	//BMS_CATL:
		(*gr_BMS_SOC						:=	gr_CATL_B2VST2SOC;
		gr_BMS_BatteryVoltage			:=	UINT_TO_REAL(gu16_CATL_B2TBMSHVVoltA);
		gr_BMS_Voltage					:=	UINT_TO_REAL(gu16_CATL_B2TBMSHVVoltA);
		//gr_BMS2_Voltage					:=	UINT_TO_REAL(gu16_CATL_B2TBMSHVVoltA);
		gs16_BMS_BatteryCurrent			:=	REAL_TO_INT(gr_CATL_B2VST2PackCurrent); 
		(*********)gu16_BMS_Maximum_Pack_Voltage	:=	REAL_TO_UINT(gr_CATL_B2VBI3PackAvaiMaxVolt); (*Limit applied to prevent overcharging*)
		gs16_BMS1_CCL					:=	REAL_TO_INT(gr_CATL_B2VAvailInpulseChrgCurr);
		gs16_BMS2_CCL					:=	REAL_TO_INT(gr_CATL_B2VAvailInpulseChrgCurr);
		//gu16_BMS_AverageCellVoltage		:=	(gu16_OrionBMS1_AverageCellVoltage + gu16_OrionBMS2_AverageCellVoltage) / 2;
		//gu16_BMS_LowCellVoltage			:=	MIN(gu16_OrionBMS1_LowCellVoltage, gu16_OrionBMS2_LowCellVoltage);
		//gu16_BMS_HighCellVoltage		:=	MAX(gu16_OrionBMS1_HighCellVoltage, gu16_OrionBMS2_HighCellVoltage);
		gr_BMS_AverageTemp				:=	INT_TO_REAL(g16_CATL_B2VST4AvgTemp);
		
		
		
		
		
	
		(*********)gu16_BMS1_LowCellmV		:=	REAL_TO_UINT(gr_CATL_B2VST5MinUcell*1000);
		//gu16_BMS2_LowCellmV		:=	gr_CATL_B2VST5MaxUcell*1000;
		(*********)gu16_BMS1_HighCellVoltage		:=	REAL_TO_UINT(gr_CATL_B2VST5MaxUcell);
		//gu16_BMS2_HighCellVoltage		:=	gu16_OrionBMS2_HighCellVoltage;
		//gu16_BMS1_LowCellVoltage_ID		:=	gu8_OrionBMS1_LowCellVoltNumber;
		//gu16_BMS2_LowCellVoltage_ID		:=	gu8_OrionBMS2_LowCellVoltNumber;
		//gu16_BMS1_HighCellVoltage_ID	:=	gu8_OrionBMS1_HighCellVoltNumber;
		//gu16_BMS2_HighCellVoltage_ID	:=	gu8_OrionBMS2_HighCellVoltNumber;	*)	
		
		
END_CASE




// First pass trigger resets charge interlock fault for plug release	
IF Main.firstPass.Q THEN
	chargeInterlockFlt := FALSE;
ELSIF gu16_OrionBMS1_FailsafeStatus.4 THEN
	chargeInterlockFlt := TRUE;
END_IF

END_PROGRAM

// Application/UserCode/Brusa/Brusa_1
(*==============================================================================================================*)
(*    Brusa charging function block calls and LED control                                                       *)
(*==============================================================================================================*)
PROGRAM Brusa_1
VAR
	Master           : BrusaControl; // Brusa charger master side
	Slave            : BrusaControl; // Brusa charger slave side
	
	LEDDem           : USINT; 
	LEDState         : BYTE;         // Case variable for LED states
	
	M_StateDem       : USINT;
	S_StateDem       : USINT;
	M_Unlock         : BOOL;
	S_Unlock         : BOOL;
	M_ErrCLr         : BOOL;
	S_ErrClr         : BOOL;
	M_ChargeStopAct  : BOOL;
	M_DCHVCurrLimMax : REAL;
	S_DCHVCurrLimMax : REAL;
	M_ACCurrLimMax   : REAL;
	S_ACCurrLimMax   : REAL;
	M_DCHVVoltLimMax : REAL;
	S_DCHVVoltLimMax : REAL;
	M_BalancingAmps  : REAL := 2;
	S_BalancingAmps  : REAL := 2;

	PulseTmr         : WORD;	
	PulseLength      : WORD := 50;    // Initialised to 500ms (50 * 10ms scans)
	Pulsing          : BOOL := FALSE;
	
	chargeStatus     : BYTE;
END_VAR
VAR CONSTANT
(*Charger statuswords =========================================================================================*)
	NLG_STATUS_CHARGE		: BYTE	:= 4;
	
(*Charger controlwords ========================================================================================*)
	NLG_CONTROL_STANDBY		: BYTE	:= 0;
	NLG_CONTROL_CHARGE		: BYTE	:= 1;
	
(*NLG LED States ==============================================================================================*)
	LED_OFF			        : BYTE	:= 0;
	LED_RED					: BYTE	:= 2;
	LED_GREEN_PULSE	        : BYTE  := 3;
	LED_GREEN				: BYTE	:= 4;
	LED_BLUE		        : BYTE	:= 8;
	LED_BLUE_GREEN_PULSE	: BYTE	:= 11;
	
(*Charge status  ==============================================================================================*)
	NOT_CONNECTED           : BYTE  := 0;
	STOPPED                 : BYTE  := 1;
	ERROR_ACTIVE            : BYTE  := 2;
	BALANCING               : BYTE  := 3;
	FULLY_CHARGED           : BYTE  := 4;
	NO_AC                   : BYTE  := 5;
	CHARGING                : BYTE  := 6;
	
END_VAR

(*==============================================================================================================*)
(*    Brusa charging function block calls                                                                       *)
(*==============================================================================================================*)
 // FreeContactor(); // Uncomment this to pulse welded contactors


Master (                Master := TRUE, // Master charger
	                 	BMS_OK := (OrionBMS1_RxConversion.Safety_OK OR OrionBMS2_RxConversion.Safety_OK),
                  CtrlPilotDet := Brusa1_Rx.S_CtrlPilotDet,
                  ProximityDet := Brusa1_Rx.S_ProximityDet,
                         Error := Brusa1_Rx.S_Err,
                         ACDet := Brusa1_Rx.S_ACDet,
               BalancingActive := OrionBMS1_RxConversion.gq_BMS1_BalActive,
                      SysState := gu8_SystemState,
                      StateAct := Brusa1_Rx.StateAct,
                        Status := Brusa1_Rx.StatusPP,
                Balancing_Amps := MAX	(2,(HMI_Rx.RAW_Pack_1_Balancing_Amps * 0.1)),
         Offset_Charge_Voltage := MAX	(4,(HMI_Rx.RAW_Pack_1_Offset_Volts    * 0.1)),
                           CCL := gs16_BMS1_CCL,
		      MaxChargingVolts := OrionBMS1_RxConversion.gr_OrionBMS1_Max_Charging_Voltage,
			     StopChargeReq := HMI_Rx.StopChargeRq,
			 ReportedMaxACCurr := Brusa1_Rx.ACCurrMaxAct_Rx,
			         CPMaxAmps := Brusa1_Rx.ACCurrMaxCP_Rx,
						   
                      StateDem => M_StateDem,
				  StopCharging => ,
                        Unlock => M_Unlock,
                 ErrorClearOut => M_ErrCLr,
                DCHVCurrLimMax => M_DCHVCurrLimMax,
                  ACCurrLimMax => M_ACCurrLimMax,
                DCHVVoltLimMax => M_DCHVVoltLimMax );
						   
						   
Slave (                 Master := FALSE, // Slave charger
	                 BMS_OK := (OrionBMS1_RxConversion.Safety_OK OR OrionBMS2_RxConversion.Safety_OK),
                  CtrlPilotDet := Brusa1_Rx.S_CtrlPilotDet,
                  ProximityDet := Brusa1_Rx.S_ProximityDet,
                         Error := Brusa2_Rx.S_Err,
                         ACDet := Brusa2_Rx.S_ACDet,
               BalancingActive := OrionBMS2_RxConversion.gq_BMS2_BalActive,
                      SysState := gu8_SystemState,
                      StateAct := Brusa2_Rx.StateAct,
                        Status := Brusa1_Rx.StatusPP,
                Balancing_Amps := MAX	(2,(HMI_Rx.RAW_Pack_2_Balancing_Amps * 0.1)),
         Offset_Charge_Voltage := MAX	(4,(HMI_Rx.RAW_Pack_2_Offset_Volts    * 0.1)),
                           CCL := gs16_BMS2_CCL,
			  MaxChargingVolts := OrionBMS2_RxConversion.gr_OrionBMS2_Max_Charging_Voltage,
			     StopChargeReq := HMI_Rx.StopChargeRq,
             ReportedMaxACCurr := Brusa2_Rx.ACCurrMaxAct_Rx,
			 	     CPMaxAmps := Brusa1_Rx.ACCurrMaxCP_Rx,
						   
                      StateDem => S_StateDem,
                        //Unlock => S_Unlock,
                 ErrorClearOut => S_ErrCLr,
                DCHVCurrLimMax => S_DCHVCurrLimMax,
                  ACCurrLimMax => S_ACCurrLimMax,
                DCHVVoltLimMax => S_DCHVVoltLimMax);	

(*==============================================================================================================*)
(*    Brusa LED control                                                                                         *)
(*==============================================================================================================*)

// Check to see if the charger is plugged in
IF (gu8_SystemState = PLUGIN_SYS) THEN    
            
	// Check for any errors
	IF (gu8_SystemState = ERROR_SYS) THEN             
		LEDDem := LED_RED;
		chargeStatus := 1;
	
	// Check for fully charged
	ELSIF gq_BattFullyCharged THEN                                                       
		LEDDem := LED_GREEN;
	
	// Check to see if charging is active
	ELSIF ((Brusa1_Rx.StateAct = NLG_STATUS_CHARGE) OR (Brusa2_Rx.StateAct = NLG_STATUS_CHARGE)) THEN
		
		// Check to see if balancing is active (Only if charging is also active)
		IF (OrionBMS1_RxConversion.gq_BMS1_BalActive OR OrionBMS2_RxConversion.gq_BMS2_BalActive) THEN
			LEDDem := LED_BLUE_GREEN_PULSE;
		ELSE
			LEDDem := LED_BLUE;
		END_IF
		
	// Check to see that AC is detected
	ELSIF NOT (Brusa1_Rx.S_ACDet) THEN
		LEDDem := LED_GREEN_PULSE; 

END_IF

ELSE 
LEDDem := 0; // OFF 

END_IF

(*==============================================================================================================*)
(*    Charge status for HMI Tx                                                                                  *)
(*==============================================================================================================*)

// System is in error state
IF (gu8_SystemState = ERROR_SYS) THEN
	chargeStatus := ERROR_ACTIVE;

// System is in plug in state (charge plug detected)
ELSIF (gu8_SystemState = PLUGIN_SYS) THEN
	
	// Charge stopped by HMI
	IF (M_ChargeStopAct) THEN
		chargeStatus := STOPPED;
	
	// Vehicle is fully charged	
	ELSIF (BMSData.Batteries_Fully_Charged AND NOT (OrionBMS1_RxConversion.gq_BMS1_BalActive OR OrionBMS2_RxConversion.gq_BMS2_BalActive)) THEN
		chargeStatus := FULLY_CHARGED;
	
	// Waiting for AC	
	ELSIF NOT (Brusa1_Rx.S_ACDet AND Brusa2_Rx.S_ACDet) THEN
		chargeStatus := NO_AC; 
	
	// BMS is balancing	
	ELSIF (OrionBMS1_RxConversion.gq_BMS1_BalActive OR OrionBMS2_RxConversion.gq_BMS2_BalActive) THEN
		chargeStatus := BALANCING;
	
	// Vehicle is charging	
	ELSIF ((Brusa1_Rx.StateAct = NLG_STATUS_CHARGE) OR (Brusa2_Rx.StateAct = NLG_STATUS_CHARGE)) THEN
		chargeStatus := CHARGING;
		
	END_IF
	
// Charge plug not detected	
ELSE
	chargeStatus := NOT_CONNECTED;

END_IF

ACTION FreeContactor:
(*==============================================================================================================*)
(*    Uncomment this action to pulse the contactor free                                                         *)
(*==============================================================================================================*)
Pulsing := TRUE;                                               // Flag to stop Contactor control from running (main())

PulseTmr := PulseTmr + 1;                                      // Increment pulse timer every scan

IF (PulseTmr = PulseLength) THEN                               // Pulse length is number of 10ms scans
DO_q_Battery1ChargeMain_DO := NOT DO_q_Battery1ChargeMain_DO;  // Switch output
PulseTmr := 0;                                                 // Reset timer
END_IF
END_ACTION

END_PROGRAM

// Application/UserCode/Brusa/BrusaControl_1
(*===================================================================================================*)
(* Charger Control                                                                                   *)
(*===================================================================================================*)
FUNCTION_BLOCK BrusaControl_1
VAR_INPUT
(*Variable inputs ===================================================================================*)
	Master                  : BOOL;             // Master?
	BMS_OK     			    : BOOL;             // Battery safety ok signal
	CtrlPilotDet            : BOOL;
	ProximityDet            : BOOL;
	Error                   : BOOL;             // Brusa error
	ACDet                   : BOOL;
	BalancingActive         : BOOL; 
	StopChargeReq           : BOOL;             // Request to stop charging
	SysState                : BYTE;             // System state
	StateAct                : BYTE;             // Brusa recieved state
	Status                  : BYTE;             // Status PP?
	Balancing_Amps          : REAL;
	OffSet_Charge_Voltage   : REAL;
	CCL                     : REAL;
	MaxChargingVolts        : REAL;             // Max charging voltage from BMS
	ReportedMaxACCurr       : WORD;             // Reported AC max current from Brusa
	CPMaxAmps               : UINT;             // Control pilot allowable current
	
	
	
END_VAR
VAR_OUTPUT
	StateDem		        : USINT;           // Charger state request
	Unlock                  : BOOL;            // Charger unlock
	ErrorClearOut           : BOOL := FALSE;   // Request error clear
	StopCharging            : BOOL;            // Latch for stop charging request
	DCHVCurrLimMax			: REAL := 0;
	ACCurrLimMax			: REAL := 0;
	DCHVVoltLimMax			: REAL := 0;

END_VAR

VAR
	ChargerStates           :	tUpdate;         // Charger state machine variable
	
	ResetCnt                :   BYTE;            // Number of reset attempts

	ChargeDelayTmr          :   WORD;            // Scan counter to delay start charging 
	
	ResetOK     			:	BOOL;            // OK to reset
	
	CurrentLimit            :   REAL;            // Maximum allowable current
			
END_VAR

VAR CONSTANT

(*Charger control words ============================================================================*)
	NLG_CONTROL_STANDBY		:	USINT	:=	0;    // Standby request
	NLG_CONTROL_CHARGE		:	USINT	:=	1;	  // Charge request
	NLG_CONTROL_SLEEP		:	USINT	:=	6;    // Sleep request
	NLG_CONTROL_SNA			:	USINT	:=	7;    
	
(*Charger status words =============================================================================*)
	NLG_STATUS_SLEEP		:	USINT	:=	0;
	NLG_STATUS_WAKEUP		:	USINT	:=	1;
	NLG_STATUS_STANDBY		:	USINT	:=	2;
	NLG_STATUS_READY2CHARGE	:	USINT	:=	3;
	NLG_STATUS_CHARGE		:	USINT	:=	4;
	NLG_STATUS_SHUTDOWN		:	USINT	:=	5;
	
(* Case step constants =============================================================================*)
	_Sleep                  :   BYTE    := 0;
	_Standby                :   BYTE 	:= 1;
	_Charging               :   BYTE    := 2;
	_Error                  :   BYTE    := 255;
	
(* Charger plug in states ==========================================================================*)
	CHARGER_DETECTED		:	BYTE	:=	0;
	CHARGER_NOTCONNECTED	:	BYTE	:=	5;
	
	PP_32A					:	BYTE	:=	3;
	PP_64A					:	BYTE	:=	4;
	
END_VAR

(*===================================================================================================*)
(* Charger state machine                                                                             *)
(*===================================================================================================*)

// Discuss error clearing - looks like error clear message is always set to false

(* Handle charge lock request =======================================================================*)	
IF (StopChargeReq) THEN                        // Move to standy if charge stop requested from HMI
	StopCharging := TRUE;
ELSIF (StopCharging AND NOT ProximityDet) THEN // Only allow charging once the charge plug has been removed and reinserted
	StopCharging := FALSE;
END_IF

CASE ChargerStates.Step OF
(* Sleep state ======================================================================================*)	
_Sleep:
	
	Unlock := TRUE;                           // Unlock charge plug

	IF (StateAct <> 0) THEN                   // Moved out of sleep state into wakeup state
		ChargerStates.Next := _Standby;       // Move to standby state 
	END_IF
	
(* Standby state ====================================================================================*)	
_Standby:
		
	Unlock := TRUE;                                          // Unlock charge plug
		
	IF OkToCharge() THEN                                     // Charging conditions OK (If charging conditions are met then lock should engage automatically)
		Unlock := FALSE;                                     // Allow charger to lock
		IF (StateAct = NLG_STATUS_READY2CHARGE) OR (StateAct = NLG_STATUS_CHARGE) THEN
		ChargerStates.Next := _Charging;                     // Move to charging state
		END_IF
	ELSIF (Error) THEN
		ChargerStates.Next := _Error;                        // Move to error state
	ELSIF (StateAct = NLG_STATUS_SLEEP) THEN
		ChargerStates.Next := _Sleep;                        // Move to sleep state
	ELSE
		StateDem :=	NLG_CONTROL_STANDBY;                     // Set STANDBY state
	END_IF
	
(* Charging state ===================================================================================*)
_Charging:
	
	StateDem :=	NLG_CONTROL_CHARGE;          // Set CHARGING state 

	IF NOT (OkToCharge()) THEN               // If not ok to charge check for errors
		
		IF (Error) THEN
			ChargerStates.Next := _Error;    // Move to error state 
		ELSE
			ChargerStates.Next := _Standby;  // Move back to standby state 
		END_IF
		
	END_IF
	
(* Error state ======================================================================================*)
_Error:

		IF (OkToReset()) THEN	
			
			ErrorClearOut := SEL((ChargerStates.Tmr < 100), FALSE, TRUE); // Request error clear
			
			IF (ChargerStates.Tmr > 6000) THEN   // 1 min - charger requires 1 min to attempt automatic recovery or temp recovery
				ResetCnt   := ResetCnt +1;       // Increment reset count
				ChargerStates.Next := _Standby;  // Move back to Standby state	
			END_IF
			
		END_IF	
	
END_CASE

(*Set the DC current limit depending on balancing status ==========================================*)
DCHVCurrLimMax := SEL( BalancingActive, CCL, MIN(CCL, Balancing_Amps));

(*Set the AC current limit based on the wire that is plugged in ===================================*)
IF (Brusa1_Rx.ACCurrMaxPP = PP_32A) THEN
	CurrentLimit	:=	MIN(15, ((CPMaxAmps/20)-1));    // Div by 200 to get single side and A from mA, then -1 for lead acid battery
ELSIF (Brusa1_Rx.ACCurrMaxPP = PP_64A) THEN
	CurrentLimit	:=	MIN(28, ((CPMaxAmps/20)-1));    // Div by 200 to get single side and A from mA, then -1 for lead acid battery
ELSE
	CurrentLimit	:=	0;
END_IF

(* Delay charge and then ramp current up to max - Add 50mA each scan ==============================*)

// If available currrent limit drops then drop requested current immediately
IF (ACCurrLimMax > CurrentLimit) THEN
	ACCurrLimMax := CurrentLimit;
	
// If available current is less than requested increase by 50mA each scan (e.g. 30Amps achieved in 6s)
ELSIF (ACCurrLimMax < CurrentLimit) THEN
	ACCurrLimMax := ACCurrLimMax + 0.005;

// Otherwise request the maximum allowable current
ELSE
	ACCurrLimMax := CurrentLimit;
END_IF

(* Limit maximum voltage to be delivered to each pack =============================================*)
DCHVVoltLimMax	:=	(MaxChargingVolts) - (OffSet_Charge_Voltage); 

Update(ADR(ChargerStates));                                     // State machine update

(*===================================================================================================*)
(* Monitor charging conditions                                                                       *)
(*===================================================================================================*)
METHOD OkToCharge : BOOL
VAR_INPUT
END_VAR
(*===================================================================================================*)
(* Monitor charging conditions                                                                       *)
(*===================================================================================================*)
OkToCharge := ((BMS_OK                                 	                               AND  // Check BMS safety is OK
              (CtrlPilotDet OR ACDet)                                                  AND  // Check for Control pilot or ACHV
	        //(ProximityDet                                                            AND  // Check plug proximity detect
			  (Status = CHARGER_DETECTED)                                              AND  // Check staus charger detected
			   NOT (Error OR StopChargeReq OR StopCharging)));                              // Check there are no errors or stop charge request
END_METHOD

(*===================================================================================================*)
(* Monitor reset conditions                                                                          *)
(*===================================================================================================*)
METHOD OkToReset : BOOL
VAR_INPUT
END_VAR
(*===================================================================================================*)
(* Monitor reset conditions                                                                          *)
(*===================================================================================================*)

OkToReset := ((StateAct = NLG_STATUS_STANDBY) AND   // Check for standby mode
			  (ResetCnt < 3));                      // Check reset count is less than 3
END_METHOD

END_FUNCTION_BLOCK

// Application/UserCode/CAN1/CAN1_Rx_1
PROGRAM CAN1_Rx_1
VAR
	Accelerator_Dennis_Rx	:	Receive_CAN1_EXD_28bit;
	Brake_Dennis_Rx			:	Receive_CAN1_EXD;
	GearSelect_Dennis_Rx	:	Receive_CAN1_EXD_28bit;
	AirPressure_Dennis_Rx	:	Receive_CAN1_EXD;
	
	EBC1_KB_Rx				:	Receive_CAN1_EXD;
	VDC1_KB_Rx				:	Receive_CAN1_EXD;
	EBC2_KB_Rx				:	Receive_CAN1_EXD;
	
	RegenStick01_Rx			:	Receive_CAN1_EXD;
	RegenStick12_Rx			:	Receive_CAN1_EXD;
	
	Bob_Handbrake_Rx	:	Receive_CAN1_EXD;
	Bob_Brake_Rx		:	Receive_CAN1_EXD;
	Bob_Accel_Rx		:	Receive_CAN1_EXD;
	Bob_RegenSelector_Rx	:	Receive_CAN1_EXD;
	
	Bob_WheelSpeed_Rx	:	Receive_CAN1_EXD_28bit;
	Bob_J1939_AirPressure_Rx	:	Receive_CAN1_EXD;
	
	Temperature_Rx		:	Receive_CAN1_EXD;
	Dennis_StabTracDisable_Rx	:	Receive_CAN1_EXD;
	
	Accelerator_Dennis_Rx_Timer	:	TON;
	Brake_Dennis_Rx_Timer		:	TON;
	GearSelect_Dennis_Rx_Timer	:	TON;
	Airpressure_Dennis_Rx_Timer	:	TON;
	
	hq_Bob_RightDrive_Compromised	: BOOL;
	hq_Bob_LeftDrive_Compromised	: BOOL;
	hq_Bob_RightFront_Compromised	: BOOL;
	hq_Bob_LeftFront_Compromised	: BOOL;
	
	Merc_AIR1_EAPU		:	Receive_CAN1_EXD;
	MercStalk_Rx: Receive_CAN1_EXD;
	Merc_Neutral_CAN1: BOOL := FALSE;
	Merc_Drive_CAN1: BOOL := FALSE;
	Merc_Reverse_CAN1: BOOL := FALSE;
	Dennis_No_Press: BOOL;
	Dennis_Up: BOOL;
	Dennis_Down: BOOL;
	LOADCTU: BOOL;
	InitialiseCounterValue: BYTE;
END_VAR

{region "Message Rx check"}
Accelerator_Dennis_Rx	(u32_COBID	:=	16#0CFF0211,
						q_NewData => ,
						au8_Data => ,
						u8_Length => 			);
				
(*Brake_Dennis_Rx	(u32_COBID	:=	16#18F0010B,
				q_NewData => ,
				au8_Data => ,
				u8_Length => 			);*)
				
GearSelect_Dennis_Rx	(u32_COBID	:=	16#0C010305,
						q_NewData => ,
						au8_Data => ,
						u8_Length => 			);
						
AirPressure_Dennis_Rx	(u32_COBID	:=	16#18FEAE30,
						q_NewData => ,
						au8_Data => ,
						u8_Length => 			);
						
EBC1_KB_Rx				(u32_COBID	:=	16#18F0010B,
						q_NewData => ,
						au8_Data => ,
						u8_Length => 			);

VDC1_KB_Rx				(u32_COBID	:=	16#18FE4F0B,
						q_NewData => ,
						au8_Data => ,
						u8_Length => 			);

EBC2_KB_Rx				(u32_COBID	:=	16#18FEBF0B,
						q_NewData => ,
						au8_Data => ,
						u8_Length => 			);
						
RegenStick01_Rx			(u32_COBID	:=	16#18F00021,
						q_NewData => ,
						au8_Data => ,
						u8_Length => 			);
							 
RegenStick12_Rx			(u32_COBID	:=	16#0C000003,
						q_NewData => ,
						au8_Data => ,
						u8_Length => 			);
							 
Bob_Handbrake_Rx(u32_COBID	:=	16#18FF0447,
			q_NewData => ,
			au8_Data => ,
			u8_Length => 			);
				 
Bob_Brake_Rx(u32_COBID	:=	16#14FF010B,
			q_NewData => ,
			au8_Data => ,
			u8_Length => 			);
				 
Bob_Accel_Rx(u32_COBID	:=	16#10F00300,
			q_NewData => ,
			au8_Data => ,
			u8_Length => 			);
				 
Bob_RegenSelector_Rx(u32_COBID	:=	16#14FF0300,
			q_NewData => ,
			au8_Data => ,
			u8_Length => 			);
				 
Bob_WheelSpeed_Rx(u32_COBID	:=	16#08FE6E0B,
			q_NewData => ,
			au8_Data => ,
			u8_Length => 			);
				 
Bob_J1939_AirPressure_Rx(u32_COBID := 16#14FEAE17,
			q_NewData => ,
			au8_Data => ,
			u8_Length => 			);
				 
Temperature_Rx(u32_COBID := 16#18FF12C4,
			q_NewData => ,
			au8_Data => ,
			u8_Length => 			);
				 
Dennis_StabTracDisable_Rx(u32_COBID := 16#18FE4F0B,
			q_NewData => ,
			au8_Data => ,
			u8_Length => 			);
				 
MercStalk_Rx	(u32_COBID	:=	16#18FF0400,
						q_NewData => ,
						au8_Data => ,
						u8_Length => 			);
(*Moved to CAN 3*)
Merc_AIR1_EAPU(u32_COBID := 16#14FEAE30,
		 	q_NewData => ,
			au8_Data => ,
			u8_Length =>			);			

{endregion}
Merc_Neutral_CAN1			:=	MercStalk_Rx.au8_Data[4].0;
Merc_Drive_CAN1				:=	MercStalk_Rx.au8_Data[4].1;
Merc_Reverse_CAN1			:=	MercStalk_Rx.au8_Data[4].2;
{region "Assign data to receive variables"}		
gu8_AccelPedal_Dennis_Rx	:=	Accelerator_Dennis_Rx.au8_Data[3];
gq_Dennis_Accel_NewData		:=	Accelerator_Dennis_Rx.q_NewData;				

gq_BrakePedal_Dennis_Rx		:=	Brake_Dennis_Rx.au8_Data[0].6;
gu8_BrakePedal_Perc_Dennis_Rx	:=	Brake_Dennis_Rx.au8_Data[1];

gu8_GearSelector_Dennis_Rx	:=	GearSelect_Dennis_Rx.au8_Data[2];
	 // Dennis Regen Select
		  
	InitialiseCounterValue := InitialiseCounterValue + 1;
	IF InitialiseCounterValue > 250 THEN
	InitialiseCounterValue := 201;
	END_IF
				   
 	IF GearSelect_Dennis_Rx.au8_Data[2] = 224 THEN
	Dennis_No_Press := TRUE;
	ELSE
	Dennis_No_Press := FALSE;
	END_IF
	
	IF GearSelect_Dennis_Rx.au8_Data[2] = 249 THEN
	Dennis_Up	:= TRUE;
	ELSE
	Dennis_Up := FALSE;
	END_IF
	
	IF GearSelect_Dennis_Rx.au8_Data[2] = 247 THEN
	Dennis_Down	:= TRUE;
	ELSE
	Dennis_Down := FALSE;
	END_IF
		 
	IF Dennis_Regen.DennisRegen.CV > 4 OR InitialiseCounterValue < 200 THEN 
	LOADCTU := TRUE;
	ELSE
	LOADCTU := FALSE;
	END_IF 
//		  
IF (AirPressure_Dennis_Rx.au8_Data[2] > 0 OR AirPressure_Dennis_Rx.au8_Data[3] > 0) THEN
	gu8_Dennis_AirPressureBrake1_Rx	:=	AirPressure_Dennis_Rx.au8_Data[2];
	gu8_Dennis_AirPressureBrake2_Rx	:=	AirPressure_Dennis_Rx.au8_Data[3];
	gu8_Dennis_AirPressureSusp_Rx	:=	AirPressure_Dennis_Rx.au8_Data[5];
END_IF

	 
gu8_EBC1_ASREngineControlActive				:=BOOL_TO_USINT(EBC1_KB_Rx.au8_Data[0].0) + SHL(BOOL_TO_USINT(EBC1_KB_Rx.au8_Data[0].1), 1);
gu8_EBC1_ASRBrakeControlActive				:=BOOL_TO_USINT(EBC1_KB_Rx.au8_Data[0].2) + SHL(BOOL_TO_USINT(EBC1_KB_Rx.au8_Data[0].3), 1);
gu8_EBC1_ABSActive							:=BOOL_TO_USINT(EBC1_KB_Rx.au8_Data[0].4) + SHL(BOOL_TO_USINT(EBC1_KB_Rx.au8_Data[0].5), 1);
gu8_EBC1_EBSBrakeSwitch						:=BOOL_TO_USINT(EBC1_KB_Rx.au8_Data[0].6) + SHL(BOOL_TO_USINT(EBC1_KB_Rx.au8_Data[0].7), 1);
gu8_EBC1_BrakePedalPosition					:=EBC1_KB_Rx.au8_Data[1];
gu8_EBC1_ABSOffroadSwitch					:=BOOL_TO_USINT(EBC1_KB_Rx.au8_Data[2].0) + SHL(BOOL_TO_USINT(EBC1_KB_Rx.au8_Data[2].1), 1);
gu8_EBC1_ASROffroadSwitch					:=BOOL_TO_USINT(EBC1_KB_Rx.au8_Data[2].2) + SHL(BOOL_TO_USINT(EBC1_KB_Rx.au8_Data[2].3), 1);
gu8_EBC1_ASRHillholderSwitch				:=BOOL_TO_USINT(EBC1_KB_Rx.au8_Data[2].4) + SHL(BOOL_TO_USINT(EBC1_KB_Rx.au8_Data[2].5), 1);
gu8_EBC1_TractionControlOverrideSwtich		:=BOOL_TO_USINT(EBC1_KB_Rx.au8_Data[2].6) + SHL(BOOL_TO_USINT(EBC1_KB_Rx.au8_Data[2].7), 1);
gu8_EBC1_AcceleratorInterlockSwitch			:=BOOL_TO_USINT(EBC1_KB_Rx.au8_Data[3].0) + SHL(BOOL_TO_USINT(EBC1_KB_Rx.au8_Data[3].1), 1);
gu8_EBC1_EngineDerateSwitch					:=BOOL_TO_USINT(EBC1_KB_Rx.au8_Data[3].2) + SHL(BOOL_TO_USINT(EBC1_KB_Rx.au8_Data[3].3), 1);
gu8_EBC1_EngineAuxiliaryShutdownSwitch		:=BOOL_TO_USINT(EBC1_KB_Rx.au8_Data[3].4) + SHL(BOOL_TO_USINT(EBC1_KB_Rx.au8_Data[3].5), 1);
gu8_EBC1_RemoteAcceleratorEnableSwitch		:=BOOL_TO_USINT(EBC1_KB_Rx.au8_Data[3].6) + SHL(BOOL_TO_USINT(EBC1_KB_Rx.au8_Data[3].7), 1);
gu8_EBC1_EngineRetarderSelection			:=EBC1_KB_Rx.au8_Data[4];
gu8_EBC1_ABSFullyOperational				:=BOOL_TO_USINT(EBC1_KB_Rx.au8_Data[5].0) + SHL(BOOL_TO_USINT(EBC1_KB_Rx.au8_Data[5].1), 1);
gu8_EBC1_gu8_EBC1_EBSRedWarningSignal		:=BOOL_TO_USINT(EBC1_KB_Rx.au8_Data[5].2) + SHL(BOOL_TO_USINT(EBC1_KB_Rx.au8_Data[5].3), 1);
gu8_EBC1_ABSEBSAmberWarningSignal			:=BOOL_TO_USINT(EBC1_KB_Rx.au8_Data[5].4) + SHL(BOOL_TO_USINT(EBC1_KB_Rx.au8_Data[5].5), 1);
gu8_EBC1_ATCASRInformationSignal			:=BOOL_TO_USINT(EBC1_KB_Rx.au8_Data[5].6) + SHL(BOOL_TO_USINT(EBC1_KB_Rx.au8_Data[5].7), 1);
gu8_EBC1_SrcAddrOfCrtllingDevForBrkCtrl		:=EBC1_KB_Rx.au8_Data[6];
gu8_EBC1_HaltBrakeSwitch					:=BOOL_TO_USINT(EBC1_KB_Rx.au8_Data[7].2) + SHL(BOOL_TO_USINT(EBC1_KB_Rx.au8_Data[7].3), 1);
gu8_EBC1_TrailerABSStatus					:=BOOL_TO_USINT(EBC1_KB_Rx.au8_Data[7].4) + SHL(BOOL_TO_USINT(EBC1_KB_Rx.au8_Data[7].5), 1);
gu8_EBC1_TractorMntdTrailerABSWarningSignal	:=BOOL_TO_USINT(EBC1_KB_Rx.au8_Data[7].6) + SHL(BOOL_TO_USINT(EBC1_KB_Rx.au8_Data[7].7), 1);

gu16_EBC2_KB_FrontAxleSpeed_Rx		:=	USINT_TO_UINT(EBC2_KB_Rx.au8_Data[0]) + SHL(USINT_TO_UINT(EBC2_KB_Rx.au8_Data[1]), 8);
gu16_EBC2_KB_FrontLeftRelSpd_Rx		:=	EBC2_KB_Rx.au8_Data[2];
gu16_EBC2_KB_FrontRightRelSpd_Rx	:=	EBC2_KB_Rx.au8_Data[3];
gu16_EBC2_KB_RearLeft1RelSpd_Rx		:=	EBC2_KB_Rx.au8_Data[4];
gu16_EBC2_KB_RearRight1RelSpd_Rx	:=	EBC2_KB_Rx.au8_Data[5];
gu16_EBC2_KB_RearLeft2RelSpd_Rx		:=	EBC2_KB_Rx.au8_Data[6];
gu16_EBC2_KB_RearRight2RelSpd_Rx	:=	EBC2_KB_Rx.au8_Data[7];

gu8_RegenStick01Pos					:=	RegenStick01_Rx.au8_Data[0];
gu8_RegenStick12Pos					:=	RegenStick12_Rx.au8_Data[0];	
	 
(*	 
VDC1_KB_Rx.au8_Data[0];
VDC1_KB_Rx.au8_Data[1];
VDC1_KB_Rx.au8_Data[2];
VDC1_KB_Rx.au8_Data[3];
VDC1_KB_Rx.au8_Data[4];
VDC1_KB_Rx.au8_Data[5];
VDC1_KB_Rx.au8_Data[6];
VDC1_KB_Rx.au8_Data[7];
*)		

gq_Bob_Handbrake_CAN	:=	Bob_Handbrake_Rx.au8_Data[0].0;
gu8_Bob_BrakePos_CAN	:=	Bob_Brake_Rx.au8_Data[1];
	
gu8_Bob_Accel_CAN		:=	Bob_Accel_Rx.au8_Data[1];
gu8_Bob_RegenSelector_CAN	:=	Bob_RegenSelector_Rx.au8_Data[4];
	
IF (Bob_WheelSpeed_Rx.au8_Data[0] <> 254 AND Bob_WheelSpeed_Rx.au8_Data[1] <> 254) THEN
	gu16_Bob_RightDrive_CAN	:=	USINT_TO_UINT(Bob_WheelSpeed_Rx.au8_Data[0]) + SHL(USINT_TO_UINT(Bob_WheelSpeed_Rx.au8_Data[1]), 8);
	hq_Bob_RightDrive_Compromised := FALSE;
ELSE
	IF (hq_Bob_LeftDrive_Compromised = FALSE) THEN
		gu16_Bob_RightDrive_CAN := gu16_Bob_LeftDrive_CAN;
	ELSIF (hq_Bob_RightFront_Compromised = FALSE) THEN
		gu16_Bob_RightDrive_CAN := gu16_Bob_RightFront_CAN;
	ELSIF (hq_Bob_LeftFront_Compromised = FALSE) THEN
		gu16_Bob_RightDrive_CAN := gu16_Bob_LeftFront_CAN;
	ELSE
		gu16_Bob_RightDrive_CAN := 0;
	END_IF
	hq_Bob_RightDrive_Compromised := TRUE;
END_IF
IF (Bob_WheelSpeed_Rx.au8_Data[2] <> 254 AND Bob_WheelSpeed_Rx.au8_Data[3] <> 254) THEN
	gu16_Bob_LeftDrive_CAN	:=	USINT_TO_UINT(Bob_WheelSpeed_Rx.au8_Data[2]) + SHL(USINT_TO_UINT(Bob_WheelSpeed_Rx.au8_Data[3]), 8);
	hq_Bob_LeftDrive_Compromised := FALSE;
ELSE
	IF (hq_Bob_RightDrive_Compromised = FALSE) THEN
		gu16_Bob_LeftDrive_CAN := gu16_Bob_RightDrive_CAN;
	ELSIF (hq_Bob_RightFront_Compromised = FALSE) THEN
		gu16_Bob_LeftDrive_CAN := gu16_Bob_RightFront_CAN;
	ELSIF (hq_Bob_LeftFront_Compromised = FALSE) THEN
		gu16_Bob_LeftDrive_CAN := gu16_Bob_LeftFront_CAN;
	ELSE
		gu16_Bob_LeftDrive_CAN := 0;
	END_IF
	hq_Bob_LeftDrive_Compromised := TRUE;
END_IF
IF (Bob_WheelSpeed_Rx.au8_Data[4] <> 254 AND Bob_WheelSpeed_Rx.au8_Data[5] <> 254) THEN
	gu16_Bob_RightFront_CAN	:=	USINT_TO_UINT(Bob_WheelSpeed_Rx.au8_Data[4]) + SHL(USINT_TO_UINT(Bob_WheelSpeed_Rx.au8_Data[5]), 8);
	hq_Bob_RightFront_Compromised := FALSE;
ELSE
	IF (hq_Bob_RightDrive_Compromised = FALSE) THEN
		gu16_Bob_RightFront_CAN := gu16_Bob_RightDrive_CAN;
	ELSIF (hq_Bob_LeftDrive_Compromised = FALSE) THEN
		gu16_Bob_RightFront_CAN := gu16_Bob_LeftDrive_CAN;
	ELSIF (hq_Bob_LeftFront_Compromised = FALSE) THEN
		gu16_Bob_RightFront_CAN := gu16_Bob_LeftFront_CAN;
	ELSE
		gu16_Bob_RightFront_CAN := 0;
	END_IF
	hq_Bob_RightFront_Compromised := TRUE;
END_IF
IF (Bob_WheelSpeed_Rx.au8_Data[6] <> 254 AND Bob_WheelSpeed_Rx.au8_Data[7] <> 254) THEN
	gu16_Bob_LeftFront_CAN	:=	USINT_TO_UINT(Bob_WheelSpeed_Rx.au8_Data[6]) + SHL(USINT_TO_UINT(Bob_WheelSpeed_Rx.au8_Data[7]), 8);
	hq_Bob_LeftFront_Compromised := FALSE;
ELSE
	IF (hq_Bob_RightDrive_Compromised = FALSE) THEN
		gu16_Bob_LeftFront_CAN := gu16_Bob_RightDrive_CAN;
	ELSIF (hq_Bob_LeftDrive_Compromised = FALSE) THEN
		gu16_Bob_LeftFront_CAN := gu16_Bob_LeftDrive_CAN;
	ELSIF (hq_Bob_RightFront_Compromised = FALSE) THEN
		gu16_Bob_LeftFront_CAN := gu16_Bob_RightFront_CAN;
	ELSE
		gu16_Bob_LeftFront_CAN := 0;
	END_IF
	hq_Bob_LeftFront_Compromised := TRUE;
END_IF
	 
IF (hq_Bob_RightDrive_Compromised = TRUE OR
	hq_Bob_LeftDrive_Compromised = TRUE OR
	hq_Bob_RightFront_Compromised = TRUE OR
	hq_Bob_LeftFront_Compromised = TRUE ) THEN

	gq_Bob_WheelSpeedSensor_Fail := TRUE;
ELSE
	gq_Bob_WheelSpeedSensor_Fail := FALSE;
END_IF

gu8_Bob_ServiceBrakeAirPressCircuit1_CAN	:=	Bob_J1939_AirPressure_Rx.au8_Data[2];
gu8_Bob_ServiceBrakeAirPressCircuit2_CAN	:=	Bob_J1939_AirPressure_Rx.au8_Data[3];
gu8_Bob_AirSuspensionSupplyPress_CAN		:=	Bob_J1939_AirPressure_Rx.au8_Data[5];
gq_Bob_AirCompressorStatus_CAN				:=	Bob_J1939_AirPressure_Rx.au8_Data[6].0;

		 
(*Temperature_Rx.au8_Data[0];*)
	 
IF (gu8_ChassisType = CHASSIS_DENNIS) THEN
	(*gq_StabTracDisable_Rx	:=	Dennis_StabTracDisable_Rx.au8_Data[0].3;*)
	gq_StabTracDisable_Rx	:=	USINT_TO_BOOL(gu8_EBC1_ASROffroadSwitch);
ELSIF (gu8_ChassisType = CHASSIS_BOB OR gu8_ChassisType = CHASSIS_ESTARGLIDER) THEN
	gq_StabTracDisable_Rx	:=	Bob_Brake_Rx.au8_Data[4].2;
END_IF
				  
{endregion}
	 
{region "Comms Loss Check"}
Accelerator_Dennis_Rx_Timer(IN := NOT(Accelerator_Dennis_Rx.q_NewData), PT := T#3S);
Brake_Dennis_Rx_Timer(IN := NOT(EBC1_KB_Rx.q_NewData), PT := T#3S);
GearSelect_Dennis_Rx_Timer(IN := NOT(GearSelect_Dennis_Rx.q_NewData), PT := T#3S);
Airpressure_Dennis_Rx_Timer(IN := NOT(Airpressure_Dennis_Rx.q_NewData), PT := T#3S);
IF (Accelerator_Dennis_Rx_Timer.Q = TRUE AND Brake_Dennis_Rx_Timer.Q = TRUE AND
	GearSelect_Dennis_Rx_Timer.Q = TRUE AND Airpressure_Dennis_Rx_Timer.Q = TRUE) THEN
	gq_Dennis_CAN1_CommsLoss	:=	TRUE;
ELSE
	gq_Dennis_CAN1_CommsLoss	:=	FALSE;
END_IF
{endregion}
	 

gu8_Merc_AirComepressor_Rq	:=	BOOL_TO_USINT(Merc_AIR1_EAPU.au8_Data[6].0) + SHL(BOOL_TO_USINT(Merc_AIR1_EAPU.au8_Data[6].1), 1);
IF ((*gu8_Merc_AirComepressor_Rq*)gq_Bob_AirCompressorStatus_CAN = TRUE(*1*)) THEN
	gq_Merc_AirComp_Rq := TRUE;
ELSE
	gq_Merc_AirComp_Rq := FALSE;
END_IF	
	 
CAN1_RxConversion();

END_PROGRAM

// Application/UserCode/CAN1/CAN1_RxConversion_1
PROGRAM CAN1_RxConversion_1
VAR
END_VAR
VAR CONSTANT
	NEUTRAL	:	USINT	:=	16#7D;
	DRIVE	:	USINT	:=	16#FC;
	REVERSE	:	USINT	:=	16#DF;
	
	AIRPRESSURE_CF	:	REAL	:=	0.08;
	
	FRONTAXLESPEED_CF	:	REAL	:=	0.00390625;
	RELATIVESPEED_CF	:	REAL	:=	0.0625;
	RELATIVESPEED_OFFSET	:	REAL	:=	-7.8125;
END_VAR


IF  gu8_GearSelector_Dennis_Rx = NEUTRAL AND gq_BrakeSwitch AND gr_VehicleSpeed_kmph <1 AND gr_VehicleSpeed_kmph >-1 THEN
	gq_Neutral_Dennis_Rq	:=	TRUE;
	gq_Drive_Dennis_Rq		:=	FALSE;
	gq_Reverse_Dennis_Rq	:=	FALSE;
ELSIF gu8_GearSelector_Dennis_Rx = DRIVE AND gq_BrakeSwitch AND gr_VehicleSpeed_kmph > -1 THEN
	gq_Neutral_Dennis_Rq	:=	FALSE;
	gq_Drive_Dennis_Rq		:=	TRUE;
	gq_Reverse_Dennis_Rq	:=	FALSE;
ELSIF gu8_GearSelector_Dennis_Rx = REVERSE AND gq_BrakeSwitch AND gr_VehicleSpeed_kmph < 1 THEN
	gq_Neutral_Dennis_Rq	:=	FALSE;
	gq_Drive_Dennis_Rq		:=	FALSE;
	gq_Reverse_Dennis_Rq	:=	TRUE;
ELSE
	;
END_IF
	
IF (gu8_EBC1_ABSActive = 1) THEN
	gq_ABSActive	:=	TRUE;
ELSE
	gq_ABSActive	:=	FALSE;
END_IF

	
gr_EBC2_KB_FrontAxleSpeed				:=	gu16_EBC2_KB_FrontAxleSpeed_Rx * FRONTAXLESPEED_CF;
gr_EBC2_KB_FrontLeftRelSpd				:=	gu16_EBC2_KB_FrontLeftRelSpd_Rx * RELATIVESPEED_CF + RELATIVESPEED_OFFSET;
gr_EBC2_KB_FrontRightRelSpd				:=	gu16_EBC2_KB_FrontRightRelSpd_Rx * RELATIVESPEED_CF + RELATIVESPEED_OFFSET;
gr_EBC2_KB_RearLeft1RelSpd				:=	gu16_EBC2_KB_RearLeft1RelSpd_Rx * RELATIVESPEED_CF + RELATIVESPEED_OFFSET;
gr_EBC2_KB_RearRight1RelSpd				:=	gu16_EBC2_KB_RearRight1RelSpd_Rx * RELATIVESPEED_CF + RELATIVESPEED_OFFSET;
gr_EBC2_KB_RearLeft2RelSpd				:=	gu16_EBC2_KB_RearLeft2RelSpd_Rx * RELATIVESPEED_CF + RELATIVESPEED_OFFSET;
gr_EBC2_KB_RearRight2RelSpd				:=	gu16_EBC2_KB_RearRight2RelSpd_Rx * RELATIVESPEED_CF + RELATIVESPEED_OFFSET;
		

gr_Bob_Accel	:=	(USINT_TO_REAL(gu8_Bob_Accel_CAN) / 250);
IF (gu8_Bob_BrakePos_CAN > 0) THEN
	gq_Bob_Brake_CAN	:=	TRUE;
ELSE
	gq_Bob_Brake_CAN	:=	FALSE;
END_IF

gr_Bob_ServiceBrakeAirPressCircuit1		:=	gu8_Bob_ServiceBrakeAirPressCircuit1_CAN * AIRPRESSURE_CF;
gr_Bob_ServiceBrakeAirPressCircuit2		:=	gu8_Bob_ServiceBrakeAirPressCircuit2_CAN * AIRPRESSURE_CF;
gr_Bob_AirSuspensionSupplyPress			:=	gu8_Bob_AirSuspensionSupplyPress_CAN * AIRPRESSURE_CF;

END_PROGRAM

// Application/UserCode/CAN1/CAN1_TCMs_Tx_1
PROGRAM CAN1_TCMs_Tx_1
VAR
	(*TCM ECR*)
	ht_RCM_C01_Tx	:	EPEC_CANVXD.Msg;
	ht_RCM_C02_Tx	:	EPEC_CANVXD.Msg;
	ht_TCM_C01_Tx	:	EPEC_CANVXD.Msg;
	ht_TCM_C02_Tx	:	EPEC_CANVXD.Msg;
	ht_TCM_C03_Tx	:	EPEC_CANVXD.Msg;
	ht_TCM_C05_Tx	:	EPEC_CANVXD.Msg;
	ht_TCM_C06_Tx	:	EPEC_CANVXD.Msg;
	ht_TCM_C08_Tx	:	EPEC_CANVXD.Msg;
	ht_TCM_C10_Tx	:	EPEC_CANVXD.Msg;
	ht_TCM_C11_Tx	:	EPEC_CANVXD.Msg;
	ht_TCM_C22_Tx	:	EPEC_CANVXD.Msg;
	ht_TCM_DM1_Tx	:	EPEC_CANVXD.Msg;
	ht_TRF1_TCM_Tx	:	EPEC_CANVXD.Msg;
	
	ht_MCM_C01_Tx	:	EPEC_CANVXD.Msg;
	ht_MCM_C02_Tx	:	EPEC_CANVXD.Msg;
	ht_MCM_C03_Tx	:	EPEC_CANVXD.Msg;
	ht_MCM_C07_Tx	:	EPEC_CANVXD.Msg;
	ht_MCM_C10_Tx	:	EPEC_CANVXD.Msg;
	ht_MCM_C14_Tx	:	EPEC_CANVXD.Msg;
	ht_MCM_C15_Tx	:	EPEC_CANVXD.Msg;
	ht_MCM_C23_Tx	:	EPEC_CANVXD.Msg;
	
	ht_Compressor_Status	:	EPEC_CANVXD.Msg;
	
	hu8_C01_Checksum	:	USINT;
	hu8_C02_Checksum	:	USINT;
	hu8_C03_Checksum	:	USINT;
	hu8_C05_Checksum	:	USINT;
	hu8_C08_Checksum	:	USINT;
	hu8_C10_Checksum	:	USINT;
	hu8_C11_Checksum	:	USINT;
	hu8_M23_Checksum	:	USINT;
	
	hu8_4BitMessageCounter10ms		:	USINT;
	hu8_4BitMessageCounter20ms		:	USINT;
	hu8_4BitMessageCounter50ms		:	USINT;
	hu8_4BitMessageCounter100ms		:	USINT;
	
	hq_CycleAlternator	:	BOOL;
	hton_MessageSend50ms_Timer	:	TON;
	hton_MessageSend_Timer		:	TON;
	Tx_Timer	:	TON;
	ClutchEnaged: BOOL;
END_VAR
VAR CONSTANT
	MAX_REGEN_TORQUE	:	UINT	:=	4090;
END_VAR
VAR
	ClutchStatB: BOOL := TRUE;
	ClutchStatA: BOOL := TRUE;
	ClutchEngaged: BOOL;
	ClutchIntermediate: BOOL;
	ClutchDisengaged: BOOL;
	TONIntermediate: TON;
END_VAR

ht_RCM_C01_Tx.ID		:=	16#CFF000F OR EPEC_CANVXD.MASK_29BIT;
ht_RCM_C01_Tx.Data[0]	:=	16#FF;
ht_RCM_C01_Tx.Data[1].0	:=	gq_RegenActive;
ht_RCM_C01_Tx.Data[1].1	:=	0;
ht_RCM_C01_Tx.Data[1].2	:=	gq_RegenActive;
ht_RCM_C01_Tx.Data[1].3	:=	0;
ht_RCM_C01_Tx.Data[1].4	:=	1;
ht_RCM_C01_Tx.Data[1].5	:=	1;
ht_RCM_C01_Tx.Data[1].6	:=	1;
ht_RCM_C01_Tx.Data[1].7	:=	1;
ht_RCM_C01_Tx.Data[2]	:=	16#FF;
ht_RCM_C01_Tx.Data[3]	:=	REAL_TO_USINT(ABS(MIN(0, gr_MCU_TorqueCommand_PreCF * BOOL_TO_USINT(gq_RegenActive) / 20))); //Should be 0 when not regenning and then a positive value when it is doing so
ht_RCM_C01_Tx.Data[4]	:=	REAL_TO_USINT(MAX_REGEN_TORQUE / 20); //Maximum regen torque is 4090Nm (MCU CAN Protocol v4.1)
ht_RCM_C01_Tx.Data[5]	:=	16#FF;
ht_RCM_C01_Tx.Data[6]	:=	16#FF;
ht_RCM_C01_Tx.Data[7]	:=	16#FF;
ht_RCM_C01_Tx.Len		:=	8;
	 
ht_RCM_C02_Tx.ID		:=	16#14FF000F OR EPEC_CANVXD.MASK_29BIT;
ht_RCM_C02_Tx.Data[0]	:=	16#FF;
ht_RCM_C02_Tx.Data[1]	:=	16#FF;
ht_RCM_C02_Tx.Data[2]	:=	16#FF;
ht_RCM_C02_Tx.Data[3]	:=	16#FF;
ht_RCM_C02_Tx.Data[4]	:=	16#FF;
ht_RCM_C02_Tx.Data[5]	:=	16#FF;
ht_RCM_C02_Tx.Data[6]	:=	16#FF;
ht_RCM_C02_Tx.Data[7]	:=	16#FF;
ht_RCM_C02_Tx.Len		:=	8;
	 
ht_TCM_C01_Tx.ID		:=	16#08FF0003 OR EPEC_CANVXD.MASK_29BIT;
ht_TCM_C01_Tx.Data[0]	:=	16#FF;
ht_TCM_C01_Tx.Data[1]	:=	16#FF;
ht_TCM_C01_Tx.Data[2]	:=	16#FF;
ht_TCM_C01_Tx.Data[3]	:=	16#FF;
ht_TCM_C01_Tx.Data[4]	:=	16#FF;
ht_TCM_C01_Tx.Data[5]	:=	16#FF;
ht_TCM_C01_Tx.Data[6].0	:=	1;
ht_TCM_C01_Tx.Data[6].1	:=	1;
ht_TCM_C01_Tx.Data[6].2	:=	1;
ht_TCM_C01_Tx.Data[6].3	:=	1;
ht_TCM_C01_Tx.Data[6].4	:=	hu8_4BitMessageCounter10ms.0;
ht_TCM_C01_Tx.Data[6].5	:=	hu8_4BitMessageCounter10ms.1;
ht_TCM_C01_Tx.Data[6].6	:=	hu8_4BitMessageCounter10ms.2;
ht_TCM_C01_Tx.Data[6].7	:=	hu8_4BitMessageCounter10ms.3;
hu8_C01_Checksum		:=	16#FF - (ht_TCM_C01_Tx.Data[0] + ht_TCM_C01_Tx.Data[1] + ht_TCM_C01_Tx.Data[2] + ht_TCM_C01_Tx.Data[3] + ht_TCM_C01_Tx.Data[4] + ht_TCM_C01_Tx.Data[5] + ht_TCM_C01_Tx.Data[6]);;
ht_TCM_C01_Tx.Data[7]	:=	hu8_C01_Checksum;
ht_TCM_C01_Tx.Len		:=	8;

ht_TCM_C02_Tx.ID		:=	16#08FF0103 OR EPEC_CANVXD.MASK_29BIT;
ht_TCM_C02_Tx.Data[0]	:=	16#FF;
ht_TCM_C02_Tx.Data[1]	:=	16#FF;
ht_TCM_C02_Tx.Data[2]	:=	UINT_TO_USINT(gu16_TCM2_OutputShaftSpeed);
ht_TCM_C02_Tx.Data[3]	:=	UINT_TO_USINT(SHR(gu16_TCM2_OutputShaftSpeed, 8));
ht_TCM_C02_Tx.Data[4]	:=	16#FF;
ht_TCM_C02_Tx.Data[5].0	:=	gu8_TCM2_DrvDirec_Stat.0;
ht_TCM_C02_Tx.Data[5].1	:=	gu8_TCM2_DrvDirec_Stat.1;
ht_TCM_C02_Tx.Data[5].2	:=	1;
ht_TCM_C02_Tx.Data[5].3	:=	1;
ht_TCM_C02_Tx.Data[5].4	:=	gu8_TCM2_RotSens_Stat.0;
ht_TCM_C02_Tx.Data[5].5	:=	gu8_TCM2_RotSens_Stat.1;
ht_TCM_C02_Tx.Data[5].6	:=	1;
ht_TCM_C02_Tx.Data[5].7	:=	1;
ht_TCM_C02_Tx.Data[6].0	:=	ClutchStatA;
ht_TCM_C02_Tx.Data[6].1	:=	ClutchStatB;
ht_TCM_C02_Tx.Data[6].2	:=	1;
ht_TCM_C02_Tx.Data[6].3	:=	1;
ht_TCM_C02_Tx.Data[6].4	:=	hu8_4BitMessageCounter10ms.0;
ht_TCM_C02_Tx.Data[6].5	:=	hu8_4BitMessageCounter10ms.1;
ht_TCM_C02_Tx.Data[6].6	:=	hu8_4BitMessageCounter10ms.2;
ht_TCM_C02_Tx.Data[6].7	:=	hu8_4BitMessageCounter10ms.3;
hu8_C02_Checksum	:=	16#FF - (ht_TCM_C02_Tx.Data[0] + ht_TCM_C02_Tx.Data[1] + ht_TCM_C02_Tx.Data[2] + ht_TCM_C02_Tx.Data[3] + ht_TCM_C02_Tx.Data[4] + ht_TCM_C02_Tx.Data[5] + ht_TCM_C02_Tx.Data[6]);
ht_TCM_C02_Tx.Data[7]	:=	hu8_C02_Checksum;
ht_TCM_C02_Tx.Len		:=	8;

ht_TCM_C03_Tx.ID		:=	16#08FF0203 OR EPEC_CANVXD.MASK_29BIT;
ht_TCM_C03_Tx.Data[0]	:=	16#FF;
ht_TCM_C03_Tx.Data[1]	:=	16#FF;
ht_TCM_C03_Tx.Data[2]	:=	UINT_TO_USINT(gu16_TCM03_ShaftSpeed_Tx);
ht_TCM_C03_Tx.Data[3]	:=	UINT_TO_USINT(SHR(gu16_TCM03_ShaftSpeed_Tx, 8));
ht_TCM_C03_Tx.Data[4]	:=	16#FF;
ht_TCM_C03_Tx.Data[5]	:=	16#FF;
ht_TCM_C03_Tx.Data[6].0	:=	1;
ht_TCM_C03_Tx.Data[6].1	:=	1;
ht_TCM_C03_Tx.Data[6].2	:=	1;
ht_TCM_C03_Tx.Data[6].3	:=	1;
ht_TCM_C03_Tx.Data[6].4	:=	hu8_4BitMessageCounter10ms.0;
ht_TCM_C03_Tx.Data[6].5	:=	hu8_4BitMessageCounter10ms.1;
ht_TCM_C03_Tx.Data[6].6	:=	hu8_4BitMessageCounter10ms.2;
ht_TCM_C03_Tx.Data[6].7	:=	hu8_4BitMessageCounter10ms.3;
hu8_C03_Checksum	:=	16#FF - (ht_TCM_C03_Tx.Data[0] + ht_TCM_C03_Tx.Data[1] + ht_TCM_C03_Tx.Data[2] + ht_TCM_C03_Tx.Data[3] + ht_TCM_C03_Tx.Data[4] + ht_TCM_C03_Tx.Data[5] + ht_TCM_C03_Tx.Data[6]);
ht_TCM_C03_Tx.Data[7]	:=	hu8_C03_Checksum;
ht_TCM_C03_Tx.Len		:=	8;

ht_TCM_C05_Tx.ID		:=	16#14FF0403 OR EPEC_CANVXD.MASK_29BIT;
ht_TCM_C05_Tx.Data[0]	:=	16#FF;
ht_TCM_C05_Tx.Data[1]	:=	16#FF;
ht_TCM_C05_Tx.Data[2]	:=	16#FF;
ht_TCM_C05_Tx.Data[3]	:=	16#FF;
ht_TCM_C05_Tx.Data[4]	:=	16#FF;
ht_TCM_C05_Tx.Data[5]	:=	16#FF;
ht_TCM_C05_Tx.Data[6].0	:=	gq_Gear_Neutral;
ht_TCM_C05_Tx.Data[6].1	:=	0;
ht_TCM_C05_Tx.Data[6].2	:=	1;
ht_TCM_C05_Tx.Data[6].3	:=	1;
ht_TCM_C05_Tx.Data[6].4	:=	hu8_4BitMessageCounter100ms.0;
ht_TCM_C05_Tx.Data[6].5	:=	hu8_4BitMessageCounter100ms.1;
ht_TCM_C05_Tx.Data[6].6	:=	hu8_4BitMessageCounter100ms.2;
ht_TCM_C05_Tx.Data[6].7	:=	hu8_4BitMessageCounter100ms.3;
hu8_C05_Checksum	:=	16#FF - (ht_TCM_C05_Tx.Data[0] + ht_TCM_C05_Tx.Data[1] + ht_TCM_C05_Tx.Data[2] + ht_TCM_C05_Tx.Data[3] + ht_TCM_C05_Tx.Data[4] + ht_TCM_C05_Tx.Data[5] + ht_TCM_C05_Tx.Data[6]);
ht_TCM_C05_Tx.Data[7]	:=	hu8_C05_Checksum;
ht_TCM_C05_Tx.Len		:=	8;

ht_TCM_C06_Tx.ID		:=	16#18FF0503 OR EPEC_CANVXD.MASK_29BIT;
ht_TCM_C06_Tx.Data[0]	:=	16#FF;
ht_TCM_C06_Tx.Data[1]	:=	16#FF;
ht_TCM_C06_Tx.Data[2]	:=	16#FF;
ht_TCM_C06_Tx.Data[3]	:=	16#FF;
ht_TCM_C06_Tx.Data[4]	:=	16#FF;
ht_TCM_C06_Tx.Data[5]	:=	16#FF;
ht_TCM_C06_Tx.Data[6]	:=	16#FF;
ht_TCM_C06_Tx.Data[7]	:=	16#FF;
ht_TCM_C06_Tx.Len		:=	8;

ht_TCM_C08_Tx.ID		:=	16#0CFF0703 OR EPEC_CANVXD.MASK_29BIT;
ht_TCM_C08_Tx.Data[0]	:=	16#FF;
ht_TCM_C08_Tx.Data[1]	:=	16#FF;
ht_TCM_C08_Tx.Data[2]	:=	16#FF;
ht_TCM_C08_Tx.Data[3]	:=	16#FF;
ht_TCM_C08_Tx.Data[4]	:=	gu8_TCM8_Gear;
ht_TCM_C08_Tx.Data[5]	:=	16#FF;
ht_TCM_C08_Tx.Data[6].0	:=	NOT(gq_Gear_Neutral);
ht_TCM_C08_Tx.Data[6].1	:=	0;
ht_TCM_C08_Tx.Data[6].2	:=	gu8_TCM8_DrvDirByGr_Stat.0;
ht_TCM_C08_Tx.Data[6].3	:=	gu8_TCM8_DrvDirByGr_Stat.1;
ht_TCM_C08_Tx.Data[6].4	:=	hu8_4BitMessageCounter20ms.0;
ht_TCM_C08_Tx.Data[6].5	:=	hu8_4BitMessageCounter20ms.1;
ht_TCM_C08_Tx.Data[6].6	:=	hu8_4BitMessageCounter20ms.2;
ht_TCM_C08_Tx.Data[6].7	:=	hu8_4BitMessageCounter20ms.3;
hu8_C08_Checksum	:=	16#FF - (ht_TCM_C08_Tx.Data[0] + ht_TCM_C08_Tx.Data[1] + ht_TCM_C08_Tx.Data[2] + ht_TCM_C08_Tx.Data[3] + ht_TCM_C08_Tx.Data[4] + ht_TCM_C08_Tx.Data[5] + ht_TCM_C08_Tx.Data[6]);
ht_TCM_C08_Tx.Data[7]	:=	hu8_C08_Checksum;
ht_TCM_C08_Tx.Len		:=	8;

ht_TCM_C10_Tx.ID		:=	16#10FF0903 OR EPEC_CANVXD.MASK_29BIT;
ht_TCM_C10_Tx.Data[0]	:=	16#FF;
ht_TCM_C10_Tx.Data[1]	:=	16#FF;
ht_TCM_C10_Tx.Data[2]	:=	16#FF;
ht_TCM_C10_Tx.Data[3]	:=	16#FF;
ht_TCM_C10_Tx.Data[4]	:=	16#FF;
ht_TCM_C10_Tx.Data[5]	:=	16#FF;
ht_TCM_C10_Tx.Data[6].0	:=	1;
ht_TCM_C10_Tx.Data[6].1	:=	1;
ht_TCM_C10_Tx.Data[6].2	:=	1;
ht_TCM_C10_Tx.Data[6].3	:=	1;
ht_TCM_C10_Tx.Data[6].4	:=	hu8_4BitMessageCounter50ms.0;
ht_TCM_C10_Tx.Data[6].5	:=	hu8_4BitMessageCounter50ms.1;
ht_TCM_C10_Tx.Data[6].6	:=	hu8_4BitMessageCounter50ms.2;
ht_TCM_C10_Tx.Data[6].7	:=	hu8_4BitMessageCounter50ms.3;
hu8_C10_Checksum	:=	16#FF - (ht_TCM_C10_Tx.Data[0] + ht_TCM_C10_Tx.Data[1] + ht_TCM_C10_Tx.Data[2] + ht_TCM_C10_Tx.Data[3] + ht_TCM_C10_Tx.Data[4] + ht_TCM_C10_Tx.Data[5] + ht_TCM_C10_Tx.Data[6]);
ht_TCM_C10_Tx.Data[7]	:=	0;
ht_TCM_C10_Tx.Len		:=	8;

ht_TCM_C11_Tx.ID		:=	16#08FF0303 OR EPEC_CANVXD.MASK_29BIT;
ht_TCM_C11_Tx.Data[0]	:=	gu8_TCM8_Gear;
ht_TCM_C11_Tx.Data[1]	:=	16#FF;
ht_TCM_C11_Tx.Data[2]	:=	16#FF;
ht_TCM_C11_Tx.Data[3]	:=	16#FF;
ht_TCM_C11_Tx.Data[4]	:=	16#FF;
ht_TCM_C11_Tx.Data[5]	:=	16#FF;
ht_TCM_C11_Tx.Data[6]	:=	UINT_TO_USINT(gu16_TCM11_ActualGearRatio);
ht_TCM_C11_Tx.Data[7]	:=	UINT_TO_USINT(SHR(gu16_TCM11_ActualGearRatio, 8));
ht_TCM_C11_Tx.Len		:=	8;

ht_TCM_C22_Tx.ID		:=	16#18FF0703 OR EPEC_CANVXD.MASK_29BIT;
ht_TCM_C22_Tx.Data[0]	:=	16#FF;
ht_TCM_C22_Tx.Data[1]	:=	16#FF;
ht_TCM_C22_Tx.Data[2]	:=	16#FF;
ht_TCM_C22_Tx.Data[3]	:=	16#FF;
ht_TCM_C22_Tx.Data[4]	:=	16#FF;
ht_TCM_C22_Tx.Data[5]	:=	16#FF;
ht_TCM_C22_Tx.Data[6]	:=	16#FF;
ht_TCM_C22_Tx.Data[7]	:=	16#FF;
ht_TCM_C22_Tx.Len		:=	8;

(*Message not sent*)
ht_TCM_DM1_Tx.ID		:=	16#10FECA03 OR EPEC_CANVXD.MASK_29BIT;
ht_TCM_DM1_Tx.Data[0]	:=	0;
ht_TCM_DM1_Tx.Data[1]	:=	0;
ht_TCM_DM1_Tx.Data[2]	:=	0;
ht_TCM_DM1_Tx.Data[3]	:=	0;
ht_TCM_DM1_Tx.Data[4]	:=	0;
ht_TCM_DM1_Tx.Data[5]	:=	0;
ht_TCM_DM1_Tx.Data[6]	:=	0;
ht_TCM_DM1_Tx.Data[7]	:=	0;
ht_TCM_DM1_Tx.Len		:=	8;

ht_TRF1_TCM_Tx.ID		:=	16#18FEF803 OR EPEC_CANVXD.MASK_29BIT;
ht_TRF1_TCM_Tx.Data[0]	:=	16#FF;
ht_TRF1_TCM_Tx.Data[1]	:=	16#FF;
ht_TRF1_TCM_Tx.Data[2]	:=	16#FF;
ht_TRF1_TCM_Tx.Data[3]	:=	16#FF;
ht_TRF1_TCM_Tx.Data[4]	:=	16#FF;
ht_TRF1_TCM_Tx.Data[5]	:=	16#FF;
ht_TRF1_TCM_Tx.Data[6]	:=	16#FF;
ht_TRF1_TCM_Tx.Data[7]	:=	16#FF;
ht_TRF1_TCM_Tx.Len		:=	8;

(*********************************************************************)
ht_MCM_C01_Tx.ID		:=	16#08FF0001 OR EPEC_CANVXD.MASK_29BIT;
ht_MCM_C01_Tx.Data[0]	:=	16#FF;
ht_MCM_C01_Tx.Data[1]	:=	16#FF;
ht_MCM_C01_Tx.Data[2]	:=	16#FF;
ht_MCM_C01_Tx.Data[3]	:=	16#FF;
ht_MCM_C01_Tx.Data[4]	:=	16#FF;
ht_MCM_C01_Tx.Data[5]	:=	16#FF;
ht_MCM_C01_Tx.Data[6]	:=	16#FF;
ht_MCM_C01_Tx.Data[7]	:=	16#FF;
ht_MCM_C01_Tx.Len		:=	8;

ht_MCM_C02_Tx.ID		:=	16#08FF0101 OR EPEC_CANVXD.MASK_29BIT; (*commented out due to already being sent*)
ht_MCM_C02_Tx.Data[0]	:=	BOOL_TO_USINT(DOS_q_BatteryDischargeMain_DO);
ht_MCM_C02_Tx.Data[1]	:=	16#FF;
ht_MCM_C02_Tx.Data[2]	:=	UINT_TO_USINT(gu16_MCM02_EngineTorque_Tx);
ht_MCM_C02_Tx.Data[3]	:=	UINT_TO_USINT(SHR(gu16_MCM02_EngineTorque_Tx, 8));
ht_MCM_C02_Tx.Data[4]	:=	UINT_TO_USINT(gu16_RPM_Display);
ht_MCM_C02_Tx.Data[5]	:=	UINT_TO_USINT(SHR(gu16_RPM_Display, 8));
ht_MCM_C02_Tx.Data[6]	:=	16#FF;
ht_MCM_C02_Tx.Data[7]	:=	16#FF;
ht_MCM_C02_Tx.Len		:=	8;

ht_MCM_C03_Tx.ID		:=	16#14FF0001 OR EPEC_CANVXD.MASK_29BIT;
ht_MCM_C03_Tx.Data[0]	:=	16#FF;
ht_MCM_C03_Tx.Data[1]	:=	16#FF;
ht_MCM_C03_Tx.Data[2]	:=	16#FF;
ht_MCM_C03_Tx.Data[3]	:=	16#FF;
ht_MCM_C03_Tx.Data[4]	:=	16#FF;
ht_MCM_C03_Tx.Data[5]	:=	16#FF;
ht_MCM_C03_Tx.Data[6]	:=	16#FF;
ht_MCM_C03_Tx.Data[7]	:=	16#FF;
ht_MCM_C03_Tx.Len		:=	8;

ht_MCM_C07_Tx.ID		:=	16#14FF0401 OR EPEC_CANVXD.MASK_29BIT;
ht_MCM_C07_Tx.Data[0]	:=	16#FF;
ht_MCM_C07_Tx.Data[1]	:=	16#FF;
ht_MCM_C07_Tx.Data[2]	:=	16#FF;
ht_MCM_C07_Tx.Data[3]	:=	16#FF;
ht_MCM_C07_Tx.Data[4]	:=	16#FF;
ht_MCM_C07_Tx.Data[5]	:=	16#FF;
ht_MCM_C07_Tx.Data[6]	:=	16#FF;
ht_MCM_C07_Tx.Data[7]	:=	16#FF;
ht_MCM_C07_Tx.Len		:=	8;

ht_MCM_C10_Tx.ID		:=	16#18FF0201 OR EPEC_CANVXD.MASK_29BIT;
ht_MCM_C10_Tx.Data[0]	:=	16#FF;
ht_MCM_C10_Tx.Data[1]	:=	16#FF;
ht_MCM_C10_Tx.Data[2]	:=	16#FF;
ht_MCM_C10_Tx.Data[3]	:=	16#FF;
ht_MCM_C10_Tx.Data[4]	:=	16#FF;
ht_MCM_C10_Tx.Data[5]	:=	16#FF;
ht_MCM_C10_Tx.Data[6]	:=	16#FF;
ht_MCM_C10_Tx.Data[7]	:=	16#FF;
ht_MCM_C10_Tx.Len		:=	8;

ht_MCM_C14_Tx.ID		:=	16#18FF0401 OR EPEC_CANVXD.MASK_29BIT;
ht_MCM_C14_Tx.Data[0]	:=	16#FF;
ht_MCM_C14_Tx.Data[1]	:=	16#FF;
ht_MCM_C14_Tx.Data[2]	:=	16#FF;
ht_MCM_C14_Tx.Data[3]	:=	16#FF;
ht_MCM_C14_Tx.Data[4]	:=	16#FF;
ht_MCM_C14_Tx.Data[5]	:=	16#FF;
ht_MCM_C14_Tx.Data[6]	:=	16#FF;
ht_MCM_C14_Tx.Data[7]	:=	16#FF;
ht_MCM_C14_Tx.Len		:=	8;

ht_MCM_C15_Tx.ID		:=	16#0CFF0001 OR EPEC_CANVXD.MASK_29BIT;
ht_MCM_C15_Tx.Data[0]	:=	16#FF;
ht_MCM_C15_Tx.Data[1]	:=	16#FF;
ht_MCM_C15_Tx.Data[2]	:=	16#FF;
ht_MCM_C15_Tx.Data[3]	:=	16#FF;
ht_MCM_C15_Tx.Data[4]	:=	16#FF;
ht_MCM_C15_Tx.Data[5]	:=	16#FF;
ht_MCM_C15_Tx.Data[6]	:=	16#FF;
ht_MCM_C15_Tx.Data[7]	:=	16#FF;
ht_MCM_C15_Tx.Len		:=	8;

ht_MCM_C23_Tx.ID		:=	16#08FF0201 OR EPEC_CANVXD.MASK_29BIT;
ht_MCM_C23_Tx.Data[0]	:=	16#FF;
ht_MCM_C23_Tx.Data[1]	:=	16#FF;
ht_MCM_C23_Tx.Data[2]	:=	16#FF;
ht_MCM_C23_Tx.Data[3]	:=	16#FF;
ht_MCM_C23_Tx.Data[4]	:=	16#FF;
ht_MCM_C23_Tx.Data[5]	:=	16#FF;
ht_MCM_C23_Tx.Data[6].0	:=	1;
ht_MCM_C23_Tx.Data[6].1	:=	1;
ht_MCM_C23_Tx.Data[6].2	:=	1;
ht_MCM_C23_Tx.Data[6].3	:=	1;
ht_MCM_C23_Tx.Data[6].4	:=	hu8_4BitMessageCounter10ms.0;
ht_MCM_C23_Tx.Data[6].5	:=	hu8_4BitMessageCounter10ms.1;
ht_MCM_C23_Tx.Data[6].6	:=	hu8_4BitMessageCounter10ms.2;
ht_MCM_C23_Tx.Data[6].7	:=	hu8_4BitMessageCounter10ms.3;
hu8_M23_Checksum	:=	16#FF - (ht_MCM_C23_Tx.Data[0] + ht_MCM_C23_Tx.Data[1] + ht_MCM_C23_Tx.Data[2] + ht_MCM_C23_Tx.Data[3] + ht_MCM_C23_Tx.Data[4] + ht_MCM_C23_Tx.Data[5] + ht_MCM_C23_Tx.Data[6]);
ht_MCM_C23_Tx.Data[7]	:=	hu8_M23_Checksum;
ht_MCM_C23_Tx.Len		:=	8;

(*Return status of the AIR1 message to inform the chassis if the compressor is on or off DAIMLER chassis
ht_Compressor_Status.ID	:=	16#14FEAE8C OR EPEC_CANVXD.MASK_29BIT;
ht_Compressor_Status.Data[0]	:=	16#FF;
ht_Compressor_Status.Data[1]	:=	16#FF;
ht_Compressor_Status.Data[2]	:=	16#FF;
ht_Compressor_Status.Data[3]	:=	16#FF;
ht_Compressor_Status.Data[4]	:=	16#FF;
ht_Compressor_Status.Data[5]	:=	16#FF;
ht_Compressor_Status.Data[6].0	:=	gq_Merc_AirComp_Enabled;
ht_Compressor_Status.Data[6].1	:=	0;
ht_Compressor_Status.Data[6].2	:=	1;
ht_Compressor_Status.Data[6].3	:=	1;
ht_Compressor_Status.Data[6].4	:=	1;
ht_Compressor_Status.Data[6].5	:=	1;
ht_Compressor_Status.Data[6].6	:=	1;
ht_Compressor_Status.Data[6].7	:=	1;
ht_Compressor_Status.Data[7]	:=	16#FF;
ht_Compressor_Status.Len	:=	8;*)


(*10ms*)
hu8_4BitMessageCounter10ms	:=	hu8_4BitMessageCounter10ms + 1;
IF (hu8_4BitMessageCounter10ms > 15) THEN
	hu8_4BitMessageCounter10ms	:=	0;
END_IF
G_CAN1_Channel.SendMessage(i_pMSG:=ADR(ht_TCM_C01_Tx));
G_CAN1_Channel.SendMessage(i_pMSG:=ADR(ht_TCM_C02_Tx));
G_CAN1_Channel.SendMessage(i_pMSG:=ADR(ht_TCM_C03_Tx));
G_CAN1_Channel.SendMessage(i_pMSG:=ADR(ht_TCM_C11_Tx));
G_CAN1_Channel.SendMessage(i_pMSG:=ADR(ht_MCM_C01_Tx));
G_CAN1_Channel.SendMessage(i_pMSG:=ADR(ht_MCM_C02_Tx));
G_CAN1_Channel.SendMessage(i_pMSG:=ADR(ht_MCM_C23_Tx));

IF (hq_CycleAlternator = TRUE) THEN
	hu8_4BitMessageCounter20ms	:=	hu8_4BitMessageCounter20ms + 1;
	IF (hu8_4BitMessageCounter20ms > 15) THEN
		hu8_4BitMessageCounter20ms	:=	0;
	END_IF
	G_CAN1_Channel.SendMessage(i_pMSG:=ADR(ht_RCM_C01_Tx));
	G_CAN1_Channel.SendMessage(i_pMSG:=ADR(ht_TCM_C08_Tx));
	G_CAN1_Channel.SendMessage(i_pMSG:=ADR(ht_MCM_C15_Tx));
END_IF
hq_CycleAlternator	:=	NOT(hq_CycleAlternator);

hton_MessageSend50ms_Timer(IN := NOT(hton_MessageSend50ms_Timer.Q), PT := T#50MS);
IF (hton_MessageSend50ms_Timer.Q = TRUE) THEN
	hu8_4BitMessageCounter50ms	:=	hu8_4BitMessageCounter50ms + 1;
	IF (hu8_4BitMessageCounter50ms > 15) THEN
		hu8_4BitMessageCounter50ms	:=	0;
	END_IF
	G_CAN1_Channel.SendMessage(i_pMSG:=ADR(ht_TCM_C10_Tx));
END_IF

hton_MessageSend_Timer(IN := NOT(hton_MessageSend_Timer.Q), PT := T#100MS);
IF (hton_MessageSend_Timer.Q = TRUE) THEN	
	hu8_4BitMessageCounter100ms	:=	hu8_4BitMessageCounter100ms + 1;
	IF (hu8_4BitMessageCounter100ms > 15) THEN
		hu8_4BitMessageCounter100ms	:=	0;
	END_IF
	G_CAN1_Channel.SendMessage(i_pMSG:=ADR(ht_RCM_C02_Tx));
	G_CAN1_Channel.SendMessage(i_pMSG:=ADR(ht_TCM_C05_Tx));
	G_CAN1_Channel.SendMessage(i_pMSG:=ADR(ht_MCM_C03_Tx));
	G_CAN1_Channel.SendMessage(i_pMSG:=ADR(ht_MCM_C07_Tx));
END_IF

Tx_Timer(IN := NOT(Tx_Timer.Q), PT := T#1000MS);
IF (Tx_Timer.Q = TRUE) THEN
	G_CAN1_Channel.SendMessage(i_pMSG:=ADR(ht_TCM_C06_Tx));
	G_CAN1_Channel.SendMessage(i_pMSG:=ADR(ht_TCM_C22_Tx));
	G_CAN1_Channel.SendMessage(i_pMSG:=ADR(ht_TRF1_TCM_Tx));
	G_CAN1_Channel.SendMessage(i_pMSG:=ADR(ht_MCM_C10_Tx));
	G_CAN1_Channel.SendMessage(i_pMSG:=ADR(ht_MCM_C14_Tx));
	
	G_CAN1_Channel.SendMessage(i_pMSG:=ADR(ht_Compressor_Status));
	
END_IF

(* Below is to alter the state of the clutch *)
IF gq_Merc_Neutral = TRUE THEN
	ClutchStatA := FALSE;
	ClutchStatB := TRUE;
	ClutchDisengaged := TRUE;
ELSE 
	ClutchDisengaged := FALSE;
END_IF

IF 	(gq_Merc_Drive OR gq_Merc_Reverse = TRUE) AND gq_BrakeSwitch THEN
	ClutchStatA := TRUE;
	ClutchStatB := FALSE;
	ClutchIntermediate := TRUE;
ELSE
	ClutchIntermediate := FALSE;
END_IF

IF (ClutchIntermediate = TRUE) THEN
	TONIntermediate (IN := TRUE, PT := T#50MS);
ELSIF (gq_Merc_Neutral = TRUE) THEN
	TONIntermediate (IN := FALSE, PT := T#0MS);
END_IF

IF 	(gq_Merc_Drive OR gq_Merc_Reverse = TRUE) AND 
	(TONIntermediate.Q = TRUE) THEN
	ClutchStatA := FALSE;
	ClutchStatB := FALSE;
	ClutchEngaged := TRUE;
ELSE
	ClutchEngaged := FALSE;
END_IF

END_PROGRAM

// Application/UserCode/CAN1/CAN1_Tx_1
PROGRAM CAN1_Tx_1
VAR
	ht_EEC1_Tx	:	EPEC_CANVXD.Msg;
	ht_EEC2_Tx	:	EPEC_CANVXD.Msg;
	ht_EEC3_Tx	:	EPEC_CANVXD.Msg;
	ht_CCSS_Tx	:	EPEC_CANVXD.Msg;
	ht_Allison_Override_Tx: EPEC_CANVXD.Msg;
	ht_SOCDash_Tx	:	EPEC_CANVXD.Msg;
	ht_TemperatureDash	:	EPEC_CANVXD.Msg;
	ht_TransmissionWarning_Bob_Tx	:	EPEC_CANVXD.Msg;
	
	hton_MessageSend_Timer	:	TON;
	hton_MessageSend1sec_Timer	:	TON;
	
	ht_Allison_ETC7_Tx	:	EPEC_CANVXD.Msg;
	ht_Allison_ProbA_Tx	:	EPEC_CANVXD.Msg;
	
	ht_SpeedDisplay_Tx	:	EPEC_CANVXD.Msg;
	ht_ExhaustAftertreatment_Tx	:	EPEC_CANVXD.Msg;
	
	ht_RearSteerActive_Tx	:	EPEC_CANVXD.Msg;
	ht_TracStabReport_Tx	:	EPEC_CANVXD.Msg;
	
	(*ht_Test	:	EPEC_CANVXD.Msg;
	hu8_TestCounter	:	USINT;
	hu8_TestChecksum	:	USINT;
	hton_TestTimer	:	TON;*)
	
	hu8_EEC1_Byte0	:	USINT;
	hu8_EEC2_Byte0	:	USINT;
	hu8_EEC2_Byte5	:	USINT;
	hu8_EEC3_Byte7	:	USINT;
END_VAR


CAN1_TxConversion();

(*Combining transmit variables into bytes*)
hu8_EEC1_Byte0	:=	(gu8_ENG_EngineTorqueMode AND 2#00001111) +
					(SHL(gu8_ENG_ActlEngPrcntTorqueHghResolution_Tx, 4) AND 2#11110000);
hu8_EEC2_Byte0	:=	(gu8_ENG_AccelPedal1LowIdleSwitch AND 2#00000011) +
					(SHL(gu8_ENG_AccelPedalKickdownSwitch, 2) AND 2#00001100) +
					(SHL(gu8_ENG_RoadSpeedLimitStatus, 4) AND 2#00110000) +
					(SHL(gu8_ENG_AccelPedal2LowIdleSwitch, 6) AND 2#11000000);
hu8_EEC2_Byte5	:=	(gu8_ENG_VehicleAccelRateLimitStatus AND 2#00000011) +
					(SHL(gu8_ENG_MomentaryEngMaxPowEnableFeedback, 2) AND 2#00001100) +
					(SHL(gu8_ENG_DPFThermalManagementActive, 4) AND 2#00110000) +
					(SHL(gu8_ENG_SCRThermalManagementActive, 6) AND 2#11000000);
hu8_EEC3_Byte7	:=	(gu8_ENG_Aftertreatment1IntakeDewPoint AND 2#00000011) +
					(SHL(gu8_ENG_Aftertreatment1ExhaustDewPoint, 2) AND 2#00001100) +
					(SHL(gu8_ENG_Aftertreatment2IntakeDewPoint, 4) AND 2#00110000) +
					(SHL(gu8_ENG_Aftertreatment2ExhaustDewPoint, 6) AND 2#11000000);

{region "KB"}
(*Set the transmit data for the messages to be sent*)
ht_EEC1_Tx.ID		:=	16#0CF00400  OR EPEC_CANVXD.MASK_29BIT;
ht_EEC1_Tx.Data[0]	:=	hu8_EEC1_Byte0;
ht_EEC1_Tx.Data[1]	:=	gu8_ENG_DriversDemandEnginePercentTorque;
ht_EEC1_Tx.Data[2]	:=	gu8_ENG_ActualEnginePercentTorque;
ht_EEC1_Tx.Data[3]	:=	UINT_TO_USINT(gu16_ENG_EngineSpeed_Tx);
ht_EEC1_Tx.Data[4]	:=	UINT_TO_USINT(SHR(gu16_ENG_EngineSpeed_Tx, 8));
ht_EEC1_Tx.Data[5]	:=	gu8_ENG_SrcAddrOfCtrllingDevForEngCtrl;
ht_EEC1_Tx.Data[6]	:=	gu8_ENG_EngineStarterMode;
ht_EEC1_Tx.Data[7]	:=	gu8_ENG_EngineDemandPercentTorque;
ht_EEC1_Tx.Len		:=	8;

ht_EEC2_Tx.ID		:=	16#0CF00300 OR EPEC_CANVXD.MASK_29BIT;
ht_EEC2_Tx.Data[0]	:=	hu8_EEC2_Byte0;
ht_EEC2_Tx.Data[1]	:=	gu8_ENG_AccelPedalPosition_Tx;
ht_EEC2_Tx.Data[2]	:=	gu8_ENG_EnginePercLoadCurrentSpeed;
ht_EEC2_Tx.Data[3]	:=	gu8_ENG_RemoteAccelPedalPosition_Tx;
ht_EEC2_Tx.Data[4]	:=	gu8_ENG_AccelPedalPosition2_Tx;
ht_EEC2_Tx.Data[5]	:=	hu8_EEC2_Byte5;
ht_EEC2_Tx.Data[6]	:=	gu8_ENG_ActualMaxAvailableEngPercTorque_Tx;
ht_EEC2_Tx.Data[7]	:=	gu8_ENG_EstimatedPumpingPercentTorque;
ht_EEC2_Tx.Len		:=	8;

ht_EEC3_Tx.ID		:=	16#18FEDF00 OR EPEC_CANVXD.MASK_29BIT;
ht_EEC3_Tx.Data[0]	:=	gu8_ENG_NominalFrictionPercTorque;
ht_EEC3_Tx.Data[1]	:=	UINT_TO_USINT(gu16_ENG_EngDesiredOperatingSpeed_Tx);
ht_EEC3_Tx.Data[2]	:=	UINT_TO_USINT(SHR(gu16_ENG_EngDesiredOperatingSpeed_Tx, 8));
ht_EEC3_Tx.Data[3]	:=	gu8_ENG_EngDesiredOperatingSpeedAsymAdjust;
ht_EEC3_Tx.Data[4]	:=	gu8_ENG_EstEngParasiticLossPercTorque;
ht_EEC3_Tx.Data[5]	:=	UINT_TO_USINT(gu16_ENG_Aftertreatment1ExhaustGasMassFlow_Tx);
ht_EEC3_Tx.Data[6]	:=	UINT_TO_USINT(SHR(gu16_ENG_Aftertreatment1ExhaustGasMassFlow_Tx, 8));
ht_EEC3_Tx.Data[7]	:=	hu8_EEC3_Byte7;
ht_EEC3_Tx.Len		:=	8;

ht_CCSS_Tx.ID		:=	16#18FEED00 OR EPEC_CANVXD.MASK_29BIT;
ht_CCSS_Tx.Data[0]	:=	gu8_ENG_MaxVehicleSpeedLimit;
ht_CCSS_Tx.Data[1]	:=	gu8_ENG_CruiseControlHighSetSpeedLimit;
ht_CCSS_Tx.Data[2]	:=	gu8_ENG_CruiseControlLowSetSpeedLimit;
ht_CCSS_Tx.Data[3]	:=	0;
ht_CCSS_Tx.Data[4]	:=	0;
ht_CCSS_Tx.Data[5]	:=	0;
ht_CCSS_Tx.Data[6]	:=	0;
ht_CCSS_Tx.Data[7]	:=	0;
ht_CCSS_Tx.Len		:=	8;
	 
(*Allison Selector Return*)
ht_Allison_ETC7_Tx.ID		:=	16#18FE4AD3 OR EPEC_CANVXD.MASK_29BIT;
ht_Allison_ETC7_Tx.Data[0]	:=	16#03;
ht_Allison_ETC7_Tx.Data[1]	:=	gu8_ETC7_TransmissionEngaged_Tx;
ht_Allison_ETC7_Tx.Data[2]	:=	16#4F;
ht_Allison_ETC7_Tx.Data[3]	:=	16#E0;
ht_Allison_ETC7_Tx.Data[4]	:=	16#FF;
ht_Allison_ETC7_Tx.Data[5]	:=	16#F3;
ht_Allison_ETC7_Tx.Data[6]	:=	16#FF;
ht_Allison_ETC7_Tx.Data[7]	:=	16#FF;
ht_Allison_ETC7_Tx.Len		:=	8;

ht_Allison_ProbA_Tx.ID		:=	16#18EF0503 OR EPEC_CANVXD.MASK_29BIT;
ht_Allison_ProbA_Tx.Data[0]	:=	16#0A;
ht_Allison_ProbA_Tx.Data[1]	:=	16#FC;
ht_Allison_ProbA_Tx.Data[2]	:=	16#00;
ht_Allison_ProbA_Tx.Data[3]	:=	16#01;
ht_Allison_ProbA_Tx.Data[4]	:=	16#23;
ht_Allison_ProbA_Tx.Data[5]	:=	16#01;
ht_Allison_ProbA_Tx.Data[6]	:=	gu8_ProbA_GearSelected_Tx;
ht_Allison_ProbA_Tx.Data[7]	:=	gu8_ProbA_GearSelected_Tx;
ht_Allison_ProbA_Tx.Len		:=	8;

ht_SpeedDisplay_Tx.ID		:=	16#18FF82C4 OR EPEC_CANVXD.MASK_29BIT;
ht_SpeedDisplay_Tx.Data[0]	:=	REAL_TO_USINT(gr_VehicleSpeed_kmph);
ht_SpeedDisplay_Tx.Data[1]	:=	0;
ht_SpeedDisplay_Tx.Data[2]	:=	0;
ht_SpeedDisplay_Tx.Data[3]	:=	0;
ht_SpeedDisplay_Tx.Data[4]	:=	0;
ht_SpeedDisplay_Tx.Data[5]	:=	0;
ht_SpeedDisplay_Tx.Data[6]	:=	0;
ht_SpeedDisplay_Tx.Data[7]	:=	0;
ht_SpeedDisplay_Tx.Len		:=	8;
	 
ht_Allison_Override_Tx.ID			:= 16#18FF0400 OR EPEC_CANVXD.MASK_29BIT;
ht_Allison_Override_Tx.Data[1]		:=	0;
ht_Allison_Override_Tx.Data[2]		:=	0;
ht_Allison_Override_Tx.Data[3]		:=	0;
ht_Allison_Override_Tx.Data[4].0	:=	gq_Gear_Neutral;
ht_Allison_Override_Tx.Data[4].1	:=	gq_Gear_Drive;
ht_Allison_Override_Tx.Data[4].2	:=	gq_Gear_Reverse;
ht_Allison_Override_Tx.Data[5]		:=	0;
ht_Allison_Override_Tx.Data[6]		:=	0;
ht_Allison_Override_Tx.Data[7]		:=	0;
ht_Allison_Override_Tx.Len			:=	8;

ht_SOCDash_Tx.ID			:=	16#18FF013D OR EPEC_CANVXD.MASK_29BIT;
ht_SOCDash_Tx.Data[0]		:=	WORD_TO_BYTE (Dennis_Regen.RegenCounterValue);
ht_SOCDash_Tx.Data[1]		:=	0;
ht_SOCDash_Tx.Data[2]		:=	0;
ht_SOCDash_Tx.Data[3]		:=	0;
ht_SOCDash_Tx.Data[4]		:=	REAL_TO_USINT(gu8_BMS_SOC * 2.4); (* What is the scale about?? Luke Matt *)
ht_SOCDash_Tx.Data[5]		:=	16#3A;
ht_SOCDash_Tx.Data[6]		:=	0;
ht_SOCDash_Tx.Data[7]		:=	0;
ht_SOCDash_Tx.Len			:=	8;
	 
ht_TemperatureDash.ID		:=	16#0 OR EPEC_CANVXD.MASK_29BIT;
ht_TemperatureDash.Data[0]	:=	0;
ht_TemperatureDash.Data[1]	:=	0;
ht_TemperatureDash.Data[2]	:=	0;
ht_TemperatureDash.Data[3]	:=	0;
ht_TemperatureDash.Data[4]	:=	0;
ht_TemperatureDash.Data[5]	:=	0;
ht_TemperatureDash.Data[6]	:=	0;
ht_TemperatureDash.Data[7]	:=	0;
ht_TemperatureDash.Len		:=	8;

ht_ExhaustAftertreatment_Tx.ID	:=	16#18FF043D OR EPEC_CANVXD.MASK_29BIT;
ht_ExhaustAftertreatment_Tx.Data[0]	:=	0;
ht_ExhaustAftertreatment_Tx.Data[1]	:=	0;
ht_ExhaustAftertreatment_Tx.Data[2]	:=	0;  
ht_ExhaustAftertreatment_Tx.Data[3]	:=	0;  
ht_ExhaustAftertreatment_Tx.Data[4]	:=	0;  
ht_ExhaustAftertreatment_Tx.Data[5]	:=	0;  
ht_ExhaustAftertreatment_Tx.Data[6]	:=	0;  
ht_ExhaustAftertreatment_Tx.Data[7]	:=	0;
ht_ExhaustAftertreatment_Tx.Len		:=	8;  
	
	 
ht_TracStabReport_Tx.ID				:=	16#18FF400B OR EPEC_CANVXD.MASK_29BIT;
ht_TracStabReport_Tx.Data[0]		:=	gu8_TractionLoss;
ht_TracStabReport_Tx.Data[1]		:=	gu8_StabilityLoss;
ht_TracStabReport_Tx.Data[2].0		:=	Driveability.SecretTractionOff;
ht_TracStabReport_Tx.Data[3]		:=	0;
ht_TracStabReport_Tx.Data[4]		:=	0;
ht_TracStabReport_Tx.Data[5]		:=	0;
ht_TracStabReport_Tx.Data[6]		:=	0;
ht_TracStabReport_Tx.Data[7]		:=	0;
ht_TracStabReport_Tx.Len			:=	8;
	 
ht_TransmissionWarning_Bob_Tx.ID		:=	16#10FF0003 OR EPEC_CANVXD.MASK_29BIT;
ht_TransmissionWarning_Bob_Tx.Data[0]	:=	16#41;
ht_TransmissionWarning_Bob_Tx.Data[1]	:=	16#48;
ht_TransmissionWarning_Bob_Tx.Data[2]	:=	0;
ht_TransmissionWarning_Bob_Tx.Data[3]	:=	0;
ht_TransmissionWarning_Bob_Tx.Data[4]	:=	0;
ht_TransmissionWarning_Bob_Tx.Data[5]	:=	0;
ht_TransmissionWarning_Bob_Tx.Data[6]	:=	0;
ht_TransmissionWarning_Bob_Tx.Data[7]	:=	0;
ht_TransmissionWarning_Bob_Tx.Len		:=	8;
		  
	 
(*ht_RearSteerActive_Tx.ID	:=	16#18FF0401 OR EPEC_CANVXD.MASK_29BIT;
ht_RearSteerActive_Tx.Data[0]		:=	16#95;
ht_RearSteerActive_Tx.Data[1]		:=	16#FF;
ht_RearSteerActive_Tx.Data[2]		:=	16#FF;
ht_RearSteerActive_Tx.Data[3]		:=	16#41;
ht_RearSteerActive_Tx.Data[4]		:=	16#FA;
ht_RearSteerActive_Tx.Data[5]		:=	16#00;
ht_RearSteerActive_Tx.Data[6]		:=	16#0F;
ht_RearSteerActive_Tx.Data[7]		:=	16#C3;
ht_RearSteerActive_Tx.Len			:=	8;

ht_RearSteerActive_Tx.ID	:=	16#18FF0801 OR EPEC_CANVXD.MASK_29BIT;
ht_RearSteerActive_Tx.Data[0]		:=	16#FF;
ht_RearSteerActive_Tx.Data[1]		:=	16#FF;	
ht_RearSteerActive_Tx.Data[2]		:=	16#FA;	
ht_RearSteerActive_Tx.Data[3]		:=	16#FA;	
ht_RearSteerActive_Tx.Data[4]		:=	16#00;	
ht_RearSteerActive_Tx.Data[5]		:=	16#00;	
ht_RearSteerActive_Tx.Data[6]		:=	16#00;	
ht_RearSteerActive_Tx.Data[7]		:=	16#00;	
ht_RearSteerActive_Tx.Len			:=	8;*)

(*
ht_Test.ID			:=	16#0CFF0203 OR EPEC_CANVXD.MASK_29BIT;
ht_Test.Data[0]		:=	16#80;
ht_Test.Data[1]		:=	16#7D;
ht_Test.Data[2]		:=	16#FF;
ht_Test.Data[3]		:=	16#FF;
ht_Test.Data[4]		:=	16#FF;
ht_Test.Data[5]		:=	16#FF;
ht_Test.Data[6]		:=	(hu8_TestCounter * 16);
CASE (hu8_TestCounter) OF
	0: hu8_TestChecksum := 112;
	1: hu8_TestChecksum := 66;
	2: hu8_TestChecksum := 20;
	3: hu8_TestChecksum := 38;
	4: hu8_TestChecksum := 184;
	5: hu8_TestChecksum := 138;
	6: hu8_TestChecksum := 220;
	7: hu8_TestChecksum := 238;
	8: hu8_TestChecksum := 123;
	9: hu8_TestChecksum := 73;
	10: hu8_TestChecksum := 31;
	11: hu8_TestChecksum := 45;
	12: hu8_TestChecksum := 179;
	13: hu8_TestChecksum := 129;
	14: hu8_TestChecksum := 215;
	15:	hu8_TestChecksum := 229;
END_CASE
ht_Test.Data[7]		:=	hu8_TestChecksum;
ht_Test.Len			:=	8;*)
	 


			   
{endregion}
	 
{region "Send Messages"}
(*Transmit these messages*)
hton_MessageSend_Timer(IN := NOT(hton_MessageSend_Timer.Q), PT := T#60MS);
IF (hton_MessageSend_Timer.Q = TRUE) THEN
	G_CAN1_Channel.SendMessage(i_pMSG:=ADR(ht_EEC1_Tx));
	G_CAN1_Channel.SendMessage(i_pMSG:=ADR(ht_EEC2_Tx));
	G_CAN1_Channel.SendMessage(i_pMSG:=ADR(ht_EEC3_Tx));
	G_CAN1_Channel.SendMessage(i_pMSG:=ADR(ht_CCSS_Tx));
		 
	G_CAN1_Channel.SendMessage(i_pMSG:=ADR(ht_Allison_ETC7_Tx));
	G_CAN1_Channel.SendMessage(i_pMSG:=ADR(ht_Allison_ProbA_Tx));
		 
	G_CAN1_Channel.SendMessage(i_pMSG:=ADR(ht_ExhaustAftertreatment_Tx));
		 
	G_CAN1_Channel.SendMessage(i_pMSG:=ADR(ht_TracStabReport_Tx));
	G_CAN1_Channel.SendMessage(i_pMSG:=ADR(ht_TransmissionWarning_Bob_Tx));  
END_IF
hton_MessageSend1sec_Timer(IN := NOT(hton_MessageSend1sec_Timer.Q), PT := T#1000MS);
IF (hton_MessageSend1sec_Timer.Q = TRUE) THEN
	G_CAN1_Channel.SendMessage(i_pMSG:=ADR(ht_SOCDash_Tx));
	G_CAN1_Channel.SendMessage(i_pMSG:=ADR(ht_RearSteerActive_Tx));
END_IF

IF (hton_MessageSend_Timer.Q = TRUE AND gq_Allison_Pad_Override = TRUE) THEN
	G_CAN1_Channel.SendMessage(i_pMSG:=ADR(ht_Allison_Override_Tx));
END_IF	 
		  
(*hton_TestTimer(IN := NOT(hton_TestTimer.Q), PT := T#50MS);
IF (hton_TestTimer.Q = TRUE) THEN
	(*hu8_TestCounter := hu8_TestCounter + 1;
	IF (hu8_TestCounter > 15) THEN
		hu8_TestCounter := 0;
	END_IF*)
	G_CAN1_Channel.SendMessage(i_pMSG:=ADR(ht_Test)); 
END_IF*)
{endregion}

END_PROGRAM

// Application/UserCode/CAN1/CAN1_TxConversion_1
PROGRAM CAN1_TxConversion_1
VAR
	RPM_READY_GAUGE	:	UINT	:=	2816; (*Minimum value needed so that rear steer will activate*)
END_VAR
VAR CONSTANT
	DRIVEENGAGED	:	USINT	:=	3;
	DRIVEDISENGAGED	:	USINT	:=	19;
	
	GEAR_DRIVE		:	USINT	:=	68;
	GEAR_REVERSE	:	USINT	:=	82;
	GEAR_NEUTRAL	:	USINT	:=	78;
	
	MCU_OPERATIONAL		:	USINT	:=	4;
END_VAR


(*Tx preconversion*)
(*EEC1*)
gr_ENG_ActlEngPrcntTorqueHghResolution		:=	0;
gr_ENG_EngineSpeed							:=	LIMIT(500, (ABS(gr_BMS_BatteryVoltage * gs16_BMS_BatteryCurrent) + 1500), 2700) (*Batt power + 1500 Lim(500->2700) * CF*);
(*EEC2*)
gr_ENG_AccelPedalPosition1					:=	gr_AccelPedal_Perc;
gr_ENG_RemoteAccelPedalPosition				:=	0;
gr_ENG_AccelPedalPosition2					:=	0;
gr_ENG_ActualMaxAvailableEngPercTorque		:=	0;
(*EEC3*)
gr_ENG_EngDesiredOperatingSpeed				:=	0;
gr_ENG_AfterTreatment1ExhaustGasMassFlow	:=	0;

(*Need to swap all the signed intergers over to unsigned so it can be processed correctly*)

(*EEC1*) (*0C FF 7D DisplayRPM Display RPM 00 FF 7D*)
gu8_ENG_EngineTorqueMode					:=	12; (*Need to define why currently no enumeration for this*)
gu8_ENG_ActlEngPrcntTorqueHghResolution_Tx	:=	REAL_TO_USINT(gr_ENG_ActlEngPrcntTorqueHghResolution);
gu8_ENG_DriversDemandEnginePercentTorque	:=	16#FF; (*Need to define this, no current enumeration*)
gu8_ENG_ActualEnginePercentTorque			:=	0;
gu16_ENG_EngineSpeed_Tx						:=	REAL_TO_UINT(gr_ENG_EngineSpeed / 0.125);
gu8_ENG_SrcAddrOfCtrllingDevForEngCtrl			:=	0;
gu8_ENG_EngineStarterMode						:=	0;
gu8_ENG_EngineDemandPercentTorque				:=	0;
(*EEC2*) (*FF FF 00 FF FF 0F 00 00*)
gu8_ENG_AccelPedal1LowIdleSwitch			:=	0;
gu8_ENG_AccelPedalKickdownSwitch			:=	0;
gu8_ENG_RoadSpeedLimitStatus				:=	0;
gu8_ENG_AccelPedal2LowIdleSwitch			:=	0;
gu8_ENG_AccelPedalPosition_Tx				:=	0;
gu8_ENG_EnginePercLoadCurrentSpeed			:=	0;
gu8_ENG_RemoteAccelPedalPosition_Tx			:=	0;
gu8_ENG_AccelPedalPosition2_Tx				:=	0;
gu8_ENG_VehicleAccelRateLimitStatus			:=	0;
gu8_ENG_MomentaryEngMaxPowEnableFeedback	:=	0;
gu8_ENG_DPFThermalManagementActive			:=	0;
gu8_ENG_SCRThermalManagementActive			:=	0;
gu8_ENG_ActualMaxAvailableEngPercTorque_Tx	:=	0;
gu8_ENG_EstimatedPumpingPercentTorque		:=	0;
(*EEC3*) (*86 40 1F 7D 7D FF FF FF*)
gu8_ENG_NominalFrictionPercTorque			:=	0;
gu16_ENG_EngDesiredOperatingSpeed_Tx		:=	0;
gu8_ENG_EngDesiredOperatingSpeedAsymAdjust	:=	0;
gu8_ENG_EstEngParasiticLossPercTorque		:=	0;
gu16_ENG_Aftertreatment1ExhaustGasMassFlow_Tx	:=	0;
gu8_ENG_Aftertreatment1IntakeDewPoint		:=	0;
gu8_ENG_Aftertreatment1ExhaustDewPoint		:=	0;
gu8_ENG_Aftertreatment2IntakeDewPoint		:=	0;
gu8_ENG_Aftertreatment2ExhaustDewPoint		:=	0;
(*CCSS*) (*FA 64 00 FF FF FF FF FF*)
gu8_ENG_MaxVehicleSpeedLimit				:=	0;
gu8_ENG_CruiseControlHighSetSpeedLimit		:=	0;
gu8_ENG_CruiseControlLowSetSpeedLimit		:=	0;
(******************************************************************************************************************************************)
(******************************************************************************************************************************************)
(*Values to send to the Allison to get it to display*)
IF (gq_Gear_Drive = TRUE OR	gq_Gear_DriveCrawl = TRUE OR gq_Gear_Reverse = TRUE OR gq_Gear_ReverseCrawl	= TRUE) THEN
	gu8_ETC7_TransmissionEngaged_Tx	:=	DRIVEENGAGED;
ELSE
	gu8_ETC7_TransmissionEngaged_Tx	:=	DRIVEDISENGAGED;
END_IF
IF (gq_Gear_Drive = TRUE OR	gq_Gear_DriveCrawl = TRUE) THEN
	gu8_ProbA_GearSelected_Tx	:=	GEAR_DRIVE;
ELSIF (gq_Gear_Reverse = TRUE OR gq_Gear_ReverseCrawl	= TRUE) THEN
	gu8_ProbA_GearSelected_Tx	:=	GEAR_REVERSE;
ELSE
	gu8_ProbA_GearSelected_Tx	:=	GEAR_NEUTRAL;
END_IF

IF (DO_q_DashboardDCDCStatus_DO = TRUE) THEN
	gu16_RPM_Display	:=	RPM_READY_GAUGE;
ELSE
	gu16_RPM_Display	:=	0;
END_IF


gu16_MCM02_EngineTorque_Tx	:=	REAL_TO_UINT(((LIMIT(-5000, gr_MCU_MotorTorqueEstimated, 5000) + 5000) / 0.2));
gu16_TCM03_ShaftSpeed_Tx	:=	REAL_TO_UINT(LIMIT(0, ABS(gr_MCU_MotorSpeed), 8000) / 0.16);

gu16_TCM2_OutputShaftSpeed	:=	REAL_TO_UINT(MIN(ABS(gr_MCU_MotorSpeed), 8000) / 0.16);
IF (gu8_MCU_State = MCU_OPERATIONAL) THEN
	gu8_TCM2_RotSens_Stat	:=	0;(*No Standstill*) (*1: Standstill, 2: Error*)
ELSE
	gu8_TCM2_RotSens_Stat	:=	3; (*SNA*)
END_IF
IF (gr_MCU_MotorSpeed >= 0) THEN
	gu8_TCM2_DrvDirec_Stat	:=	0; //FWD
ELSE
	gu8_TCM2_DrvDirec_Stat	:=	1; //BWD
END_IF

IF (gq_Gear_Drive = TRUE) THEN
	gu8_TCM8_Gear	:=	126;
	gu8_TCM8_DrvDirByGr_Stat	:=	2;
ELSIF (gq_Gear_Reverse = TRUE) THEN
	gu8_TCM8_Gear	:=	124;
	gu8_TCM8_DrvDirByGr_Stat	:=	0;
ELSE
	gu8_TCM8_Gear	:=	125;
	gu8_TCM8_DrvDirByGr_Stat	:=	1;
END_IF

gu16_TCM11_ActualGearRatio	:=	((gu16_GearRatio_PreCF / 1000) + 25) * 1000;

END_PROGRAM

// Application/UserCode/CAN1/KB_Tx_1
PROGRAM KB_Tx_1
VAR
	ht_ETC1_Tx		:	EPEC_CANVXD.Msg;
	ht_ETC2_Tx		:	EPEC_CANVXD.Msg;
	ht_ETC8_Tx		:	EPEC_CANVXD.Msg;
	ht_ERC1_RD_Tx	:	EPEC_CANVXD.Msg;
	ht_ERC1_RE_Tx	:	EPEC_CANVXD.Msg;
	ht_RC_RD_Tx		:	EPEC_CANVXD.Msg;
	ht_RC_RE_Tx		:	EPEC_CANVXD.Msg;
	ht_TD_Tx		:	EPEC_CANVXD.Msg;
	ht_Prop37_Tx	:	EPEC_CANVXD.Msg;
	ht_Prop40_Tx	:	EPEC_CANVXD.Msg;
	ht_Prop87_Tx	:	EPEC_CANVXD.Msg;
	
	hton_MessageSend_Timer	:	TON;
	hton_TD_Timer			:	TON;
END_VAR

ht_ETC1_Tx.ID		:=	16#0CF00203 OR EPEC_CANVXD.MASK_29BIT;
ht_ETC1_Tx.Data[0]	:=	16#3D;
ht_ETC1_Tx.Data[1]	:=	16#00;
ht_ETC1_Tx.Data[2]	:=	16#00;
ht_ETC1_Tx.Data[3]	:=	16#00;
ht_ETC1_Tx.Data[4]	:=	16#00;
ht_ETC1_Tx.Data[5]	:=	16#00;
ht_ETC1_Tx.Data[6]	:=	16#00;
ht_ETC1_Tx.Data[7]	:=	16#00;
ht_ETC1_Tx.Len		:=	8;
	 
ht_ETC2_Tx.ID		:=	16#18F00503 OR EPEC_CANVXD.MASK_29BIT;
ht_ETC2_Tx.Data[0]	:=	gu8_CurrentGear2; (*Current Gear2*)
ht_ETC2_Tx.Data[1]	:=	UINT_TO_USINT(gu16_CurrentGear); (*Current Gear LSB*)
ht_ETC2_Tx.Data[2]	:=	UINT_TO_USINT(SHR(gu16_CurrentGear, 8)); (*Current Gear MSB*)
ht_ETC2_Tx.Data[3]	:=	gu8_CurrentGear2; (*Current Gear2*)
ht_ETC2_Tx.Data[4]	:=	16#FF;
ht_ETC2_Tx.Data[5]	:=	16#FF;
ht_ETC2_Tx.Data[6]	:=	UINT_TO_USINT(gu16_CurrentGear1); (*Current Gear1 LSB*)
ht_ETC2_Tx.Data[7]	:=	UINT_TO_USINT(SHR(gu16_CurrentGear1, 8)); (*Current Gear1 MSB*)
ht_ETC2_Tx.Len		:=	8;

ht_ETC8_Tx.ID		:=	16#0CF00C03 OR EPEC_CANVXD.MASK_29BIT;
ht_ETC8_Tx.Data[0]	:=	16#FF;
ht_ETC8_Tx.Data[1]	:=	16#FF;
ht_ETC8_Tx.Data[2]	:=	16#FF;
ht_ETC8_Tx.Data[3]	:=	16#FF;
ht_ETC8_Tx.Data[4]	:=	16#FF;
ht_ETC8_Tx.Data[5]	:=	16#FF;
ht_ETC8_Tx.Data[6]	:=	16#FF;
ht_ETC8_Tx.Data[7]	:=	16#FF;
ht_ETC8_Tx.Len		:=	8;

ht_ERC1_RD_Tx.ID		:=	16#18F00010 OR EPEC_CANVXD.MASK_29BIT;
ht_ERC1_RD_Tx.Data[0]	:=	16#00;
ht_ERC1_RD_Tx.Data[1]	:=	16#00;
ht_ERC1_RD_Tx.Data[2]	:=	16#00;
ht_ERC1_RD_Tx.Data[3]	:=	16#00;
ht_ERC1_RD_Tx.Data[4]	:=	16#00;
ht_ERC1_RD_Tx.Data[5]	:=	16#00;
ht_ERC1_RD_Tx.Data[6]	:=	16#00;
ht_ERC1_RD_Tx.Data[7]	:=	16#A5;
ht_ERC1_RD_Tx.Len		:=	8;

ht_ERC1_RE_Tx.ID		:=	16#18F0000F OR EPEC_CANVXD.MASK_29BIT;
ht_ERC1_RE_Tx.Data[0]	:=	16#00;
ht_ERC1_RE_Tx.Data[1]	:=	16#A5;
ht_ERC1_RE_Tx.Data[2]	:=	16#00;
ht_ERC1_RE_Tx.Data[3]	:=	16#00;
ht_ERC1_RE_Tx.Data[4]	:=	16#00;
ht_ERC1_RE_Tx.Data[5]	:=	16#00;
ht_ERC1_RE_Tx.Data[6]	:=	16#00;
ht_ERC1_RE_Tx.Data[7]	:=	16#A5;
ht_ERC1_RE_Tx.Len		:=	8;

ht_RC_RD_Tx.ID		:=	16#18FEE110 OR EPEC_CANVXD.MASK_29BIT;
ht_RC_RD_Tx.Data[0]	:=	16#00;
ht_RC_RD_Tx.Data[1]	:=	16#10;
ht_RC_RD_Tx.Data[2]	:=	16#00;
ht_RC_RD_Tx.Data[3]	:=	16#00;
ht_RC_RD_Tx.Data[4]	:=	16#00;
ht_RC_RD_Tx.Data[5]	:=	16#00;
ht_RC_RD_Tx.Data[6]	:=	16#00;
ht_RC_RD_Tx.Data[7]	:=	16#00;
ht_RC_RD_Tx.Len		:=	8;

ht_RC_RE_Tx.ID		:=	16#18FEE10F OR EPEC_CANVXD.MASK_29BIT;
ht_RC_RE_Tx.Data[0]	:=	16#00;
ht_RC_RE_Tx.Data[1]	:=	16#00;
ht_RC_RE_Tx.Data[2]	:=	16#FF;
ht_RC_RE_Tx.Data[3]	:=	16#FF;
ht_RC_RE_Tx.Data[4]	:=	16#FF;
ht_RC_RE_Tx.Data[5]	:=	16#FF;
ht_RC_RE_Tx.Data[6]	:=	16#FF;
ht_RC_RE_Tx.Data[7]	:=	16#FF;
ht_RC_RE_Tx.Len		:=	8;

ht_TD_Tx.ID			:=	16#18FEE617 OR EPEC_CANVXD.MASK_29BIT;
ht_TD_Tx.Data[0]	:=	16#FF;
ht_TD_Tx.Data[1]	:=	16#FF;
ht_TD_Tx.Data[2]	:=	16#FF;
ht_TD_Tx.Data[3]	:=	16#FF;
ht_TD_Tx.Data[4]	:=	16#FF;
ht_TD_Tx.Data[5]	:=	16#FF;
ht_TD_Tx.Data[6]	:=	16#00;
ht_TD_Tx.Data[7]	:=	16#00;
ht_TD_Tx.Len		:=	8;

ht_Prop37_Tx.ID			:=	16#0CFF2537 OR EPEC_CANVXD.MASK_29BIT;
ht_Prop37_Tx.Data[0]	:=	16#FF;
ht_Prop37_Tx.Data[1]	:=	16#FF;
ht_Prop37_Tx.Data[2]	:=	16#00;
ht_Prop37_Tx.Data[3]	:=	16#00;
ht_Prop37_Tx.Data[4]	:=	16#00;
ht_Prop37_Tx.Data[5]	:=	16#00;
ht_Prop37_Tx.Data[6]	:=	16#00;
ht_Prop37_Tx.Data[7]	:=	16#FC;
ht_Prop37_Tx.Len		:=	8;

ht_Prop40_Tx.ID			:=	16#0CFF2817 OR EPEC_CANVXD.MASK_29BIT;
ht_Prop40_Tx.Data[0]	:=	16#FC;
ht_Prop40_Tx.Data[1]	:=	16#F3;
ht_Prop40_Tx.Data[2]	:=	16#FF;
ht_Prop40_Tx.Data[3]	:=	16#00;
ht_Prop40_Tx.Data[4]	:=	16#00;
ht_Prop40_Tx.Data[5]	:=	16#00;
ht_Prop40_Tx.Data[6]	:=	16#00;
ht_Prop40_Tx.Data[7]	:=	16#00;
ht_Prop40_Tx.Len		:=	8;

ht_Prop87_Tx.ID			:=	16#0CFF5730 OR EPEC_CANVXD.MASK_29BIT;
ht_Prop87_Tx.Data[0]	:=	16#FF;
ht_Prop87_Tx.Data[1]	:=	16#FD;
ht_Prop87_Tx.Data[2]	:=	16#00;
ht_Prop87_Tx.Data[3]	:=	16#00;
ht_Prop87_Tx.Data[4]	:=	16#00;
ht_Prop87_Tx.Data[5]	:=	16#00;
ht_Prop87_Tx.Data[6]	:=	16#00;
ht_Prop87_Tx.Data[7]	:=	16#00;
ht_Prop87_Tx.Len		:=	8;




hton_MessageSend_Timer(IN := NOT(hton_MessageSend_Timer.Q), PT := T#80MS);
IF (hton_MessageSend_Timer.Q = TRUE) THEN
	G_CAN1_Channel.SendMessage(i_pMSG:=ADR(ht_ETC1_Tx));
	G_CAN1_Channel.SendMessage(i_pMSG:=ADR(ht_ETC2_Tx));
	G_CAN1_Channel.SendMessage(i_pMSG:=ADR(ht_ETC8_Tx));
	G_CAN1_Channel.SendMessage(i_pMSG:=ADR(ht_ERC1_RD_Tx));
	G_CAN1_Channel.SendMessage(i_pMSG:=ADR(ht_ERC1_RE_Tx));
	G_CAN1_Channel.SendMessage(i_pMSG:=ADR(ht_RC_RD_Tx));
	G_CAN1_Channel.SendMessage(i_pMSG:=ADR(ht_RC_RE_Tx));
	G_CAN1_Channel.SendMessage(i_pMSG:=ADR(ht_Prop37_Tx));
	G_CAN1_Channel.SendMessage(i_pMSG:=ADR(ht_Prop40_Tx));
	G_CAN1_Channel.SendMessage(i_pMSG:=ADR(ht_Prop87_Tx));
END_IF

hton_TD_Timer(IN := NOT(hton_TD_Timer.Q), PT := T#10000MS);
IF (hton_TD_Timer.Q = TRUE) THEN
	G_CAN1_Channel.SendMessage(i_pMSG:=ADR(ht_TD_Tx));
END_IF

END_PROGRAM

// Application/UserCode/CAN3/CAN3_Rx_1
PROGRAM CAN3_Rx_1
VAR
	GearSelect_Bob_Rx	:	Receive_CAN3_EXD_28bit;
	MercStalk_Rx		:	Receive_CAN3_EXD;
	Merc_AIR1_EAPU: Receive_CAN3_EXD;
	Mode_Button: BOOL;
	Up_Button: BOOL;
	Down_Button: BOOL;
END_VAR


GearSelect_Bob_Rx	(u32_COBID	:=	16#0C010305,
						q_NewData => ,
						au8_Data => ,
						u8_Length => 			);
						
MercStalk_Rx	(u32_COBID	:=	16#18FF0400,
						q_NewData => ,
						au8_Data => ,
						u8_Length => 			);
(*COPIED FROM CAN 1*)					
Merc_AIR1_EAPU	(u32_COBID := 16#14FEAE30,
		 	q_NewData => ,
			au8_Data => ,
			u8_Length =>			);	
			
IF GearSelect_Bob_Rx.au8_Data[5] = 16#7F THEN
	Mode_Button := TRUE;
ELSE
	Mode_Button := FALSE;
	END_IF

IF GearSelect_Bob_Rx.au8_Data[2] = 16#F9 THEN
	Up_Button := TRUE;
ELSE
	Up_Button := FALSE;
	END_IF

IF GearSelect_Bob_Rx.au8_Data[2] = 16#F7 THEN
	Down_Button := TRUE;
ELSE
	Down_Button := FALSE;
	END_IF
	
(*gu8_Merc_AirComepressor_Rq	:=	BOOL_TO_USINT(Merc_AIR1_EAPU.au8_Data[6].0) + SHL(BOOL_TO_USINT(Merc_AIR1_EAPU.au8_Data[6].1), 1);
IF (gu8_Merc_AirComepressor_Rq = 1) THEN 
	gq_Merc_AirComp_Rq := TRUE;
ELSE
	gq_Merc_AirComp_Rq := FALSE;
END_IF*)

(******)					
gu8_GearSelector_Bob_Rx	:=	GearSelect_Bob_Rx.au8_Data[2];

gu8_Merc_AutoManualSwitch	:=	BOOL_TO_USINT(MercStalk_Rx.au8_Data[0].0) + SHL(BOOL_TO_USINT(MercStalk_Rx.au8_Data[0].1), 1);
(*MercStalk_Rx.au8_Data[0];
MercStalk_Rx.au8_Data[1];*)
gu8_Merc_GearSelectSwitch	:=	BOOL_TO_USINT(MercStalk_Rx.au8_Data[2].2) + SHL(BOOL_TO_USINT(MercStalk_Rx.au8_Data[2].3), 1) +
								SHL(BOOL_TO_USINT(MercStalk_Rx.au8_Data[2].4), 2) + SHL(BOOL_TO_USINT(MercStalk_Rx.au8_Data[2].5), 3);
(*MercStalk_Rx.au8_Data[2];
MercStalk_Rx.au8_Data[3];*)
gq_Merc_Neutral				:=	MercStalk_Rx.au8_Data[4].0;
gq_Merc_Drive				:=	MercStalk_Rx.au8_Data[4].1;
gq_Merc_Reverse				:=	MercStalk_Rx.au8_Data[4].2;
(*MercStalk_Rx.au8_Data[4];
MercStalk_Rx.au8_Data[5];
MercStalk_Rx.au8_Data[6];
MercStalk_Rx.au8_Data[7];*)

CAN3_RxConversion();

END_PROGRAM

// Application/UserCode/CAN3/CAN3_RxConversion_1
PROGRAM CAN3_RxConversion_1
VAR
	;
END_VAR
VAR CONSTANT
	NEUTRAL	:	USINT	:=	16#7D;
	DRIVE	:	USINT	:=	16#FC;
	REVERSE	:	USINT	:=	16#DF;
	NOPRESS	:	USINT	:=	16#7C;
END_VAR



IF (gu8_GearSelector_Bob_Rx = NEUTRAL) AND (gu8_GearSelector_Bob_Rx <> 224) AND gq_BrakeSwitch = TRUE AND gr_VehicleSpeed_kmph <0.001 AND gr_VehicleSpeed_kmph >-0.001 THEN
	gq_Neutral_Bob_Rq	:=	TRUE;
	gq_Drive_Bob_Rq		:=	FALSE;
	gq_Reverse_Bob_Rq	:=	FALSE;
ELSIF (gu8_GearSelector_Bob_Rx = DRIVE) AND (gu8_GearSelector_Bob_Rx <> 224) AND gq_BrakeSwitch = TRUE AND gr_VehicleSpeed_kmph > -0.001 THEN
	gq_Neutral_Bob_Rq	:=	FALSE;
	gq_Drive_Bob_Rq		:=	TRUE;
	gq_Reverse_Bob_Rq	:=	FALSE;
ELSIF (gu8_GearSelector_Bob_Rx = REVERSE) AND (gu8_GearSelector_Bob_Rx <> 224) AND gq_BrakeSwitch = TRUE AND gr_VehicleSpeed_kmph < 0.001 THEN
	gq_Neutral_Bob_Rq	:=	FALSE;
	gq_Drive_Bob_Rq		:=	FALSE;
	gq_Reverse_Bob_Rq	:=	TRUE;
ELSE
	;
END_IF

END_PROGRAM

// Application/UserCode/CAN3/CAN3_Tx_1
PROGRAM CAN3_Tx_1
VAR
	ht_Bob_Allison_ETC7_Tx		:	EPEC_CANVXD.Msg;
	ht_Allison_Override_Tx: EPEC_CANVXD.Msg;
	ht_Bob_Allison_ProbA_Tx		:	EPEC_CANVXD.Msg;
	hton_MessageSend_Timer		:	TON;
END_VAR



(*Allison Selector Return*)
ht_Bob_Allison_ETC7_Tx.ID		:=	16#18FE4AD3 OR EPEC_CANVXD.MASK_29BIT;
ht_Bob_Allison_ETC7_Tx.Data[0]	:=	16#03;
ht_Bob_Allison_ETC7_Tx.Data[1]	:=	gu8_ETC7_TransmissionEngaged_Tx;
ht_Bob_Allison_ETC7_Tx.Data[2]	:=	16#4F;
ht_Bob_Allison_ETC7_Tx.Data[3]	:=	16#E0;
ht_Bob_Allison_ETC7_Tx.Data[4]	:=	16#FF;
ht_Bob_Allison_ETC7_Tx.Data[5]	:=	16#F3;
ht_Bob_Allison_ETC7_Tx.Data[6]	:=	16#FF;
ht_Bob_Allison_ETC7_Tx.Data[7]	:=	16#FF;
ht_Bob_Allison_ETC7_Tx.Len		:=	8;

ht_Bob_Allison_ProbA_Tx.ID		:=	16#18EF0503 OR EPEC_CANVXD.MASK_29BIT;
ht_Bob_Allison_ProbA_Tx.Data[0]	:=	16#0A;
ht_Bob_Allison_ProbA_Tx.Data[1]	:=	16#FC;
ht_Bob_Allison_ProbA_Tx.Data[2]	:=	16#00;
ht_Bob_Allison_ProbA_Tx.Data[3]	:=	16#01;
ht_Bob_Allison_ProbA_Tx.Data[4]	:=	16#23;
ht_Bob_Allison_ProbA_Tx.Data[5]	:=	16#01;
ht_Bob_Allison_ProbA_Tx.Data[6]	:=	gu8_ProbA_GearSelected_Tx;
ht_Bob_Allison_ProbA_Tx.Data[7]	:=	gu8_ProbA_GearSelected_Tx;
ht_Bob_Allison_ProbA_Tx.Len		:=	8;

ht_Allison_Override_Tx.ID		:= 16#18FF0400 OR EPEC_CANVXD.MASK_29BIT;
(*ht_Allison_Override_Tx.Data[0]	:=
ht_Allison_Override_Tx.Data[1]	:=
ht_Allison_Override_Tx.Data[2]	:=
ht_Allison_Override_Tx.Data[3]	:=*)
ht_Allison_Override_Tx.Data[4].0	:=	gq_Gear_Neutral;
ht_Allison_Override_Tx.Data[4].1	:=	gq_Gear_Drive;
ht_Allison_Override_Tx.Data[4].2	:=	gq_Gear_Reverse;
(*ht_Allison_Override_Tx.Data[5]	:=
ht_Allison_Override_Tx.Data[6]	:=
ht_Allison_Override_Tx.Data[7]	:=*)
ht_Allison_Override_Tx.Len		:=	8;

(*Transmit these messages*)
hton_MessageSend_Timer(IN := NOT(hton_MessageSend_Timer.Q), PT := T#100MS);
IF (hton_MessageSend_Timer.Q = TRUE) THEN
	G_CAN3_Channel.SendMessage(i_pMSG:=ADR(ht_Bob_Allison_ETC7_Tx));
	G_CAN3_Channel.SendMessage(i_pMSG:=ADR(ht_Bob_Allison_ProbA_Tx));
END_IF

IF (hton_MessageSend_Timer.Q = TRUE AND gq_Allison_Pad_Override = TRUE) THEN
	G_CAN3_Channel.SendMessage(i_pMSG:=ADR(ht_Allison_Override_Tx));
END_IF

END_PROGRAM

// Application/UserCode/CAN4/CAN4_Rx_1
PROGRAM CAN4_Rx_1
VAR
	Handbrake_Rx	:	Receive_CAN4_EXD;
	Handbrake_Rx_Timer	:	TON;
	
	
	
	
	
	
END_VAR

Handbrake_Rx(u32_COBID	:=	16#18FEF1F2,
			q_NewData => ,
			au8_Data => ,
			u8_Length => 			);
			
				
gq_Handbrake_CAN	:=	Handbrake_Rx.au8_Data[0].2;				
				
Handbrake_Rx_Timer(IN := NOT(Handbrake_Rx.q_NewData), PT := t#10s);

END_PROGRAM

// Application/UserCode/CAN4/CAN4_Tx_1
PROGRAM CAN4_Tx_1
VAR
	ht_CAN4_601_Tx			:	EPEC_CANVXD.Msg;
	ht_CAN4_201_Tx			:	EPEC_CANVXD.Msg;
	ht_CAN4_301_Tx			:	EPEC_CANVXD.Msg;
	ht_CAN4_401_Tx			:	EPEC_CANVXD.Msg;
	ht_CAN4_8DD1_Tx			: 	EPEC_CANVXD.Msg;
	CAN4_HMI_Tx	    		: 	EPEC_CANVXD.Msg;
	hton_MessageSend_Timer	:	TON;
	ht_ETC2_Tx				:	EPEC_CANVXD.Msg;
	NMT1_Tx					:	EPEC_CANVXD.Msg;
	Dash_FF02_Tx 			:	EPEC_CANVXD.Msg;
	Dash_FF04_Tx 			:	EPEC_CANVXD.Msg;
	Dash_FF08_Tx			:	EPEC_CANVXD.Msg;
	Dash_FF12_Tx			:	EPEC_CANVXD.Msg;
	Dash_FF14_Tx			:	EPEC_CANVXD.Msg;
	Dash_FF21_Tx			:	EPEC_CANVXD.Msg;
	Tx_Timer				:	TON;
	hu8_Temp				:	USINT := 10;
	Version					: 	STRING;
END_VAR

CAN4_TxConversion();
BMS_to_HMI();
DCDC_to_HMI();
MCU_to_HMI();
Sevcon_to_HMI();
vmu_to_hmi();
IF CAN4_TxConversion.gq_CAN4_ChargerPP_Tx THEN BRUSA_to_HMI();
END_IF
Version := Project_Infomation.ver;
 
//* special needs for HMI
ht_CAN4_8DD1_Tx.ID		:=	16#188000DD OR EPEC_CANVXD.MASK_29BIT;
ht_CAN4_8DD1_Tx.Data[0]	:=	gu8_ChassisType;
ht_CAN4_8DD1_Tx.Data[1].0	:=	gq_Frosty_NoWheelSpeedSensors;
ht_CAN4_8DD1_Tx.Data[1].1	:=	gq_BodyStepInstalled;
ht_CAN4_8DD1_Tx.Data[1].2	:=	gq_Daimler_PowerShift_Installed;
ht_CAN4_8DD1_Tx.Data[1].3	:=	gq_APU_Installed;
ht_CAN4_8DD1_Tx.Data[1].4	:=	gq_RearSteer_Installed;
ht_CAN4_8DD1_Tx.Data[1].5	:=	gq_CAN1_Merc_Gears;
ht_CAN4_8DD1_Tx.Data[1].6	:=	E_Stop_Installed;
ht_CAN4_8DD1_Tx.Data[1].7	:=	DO_q_HeaterOut_DI;
ht_CAN4_8DD1_Tx.Data[2] 	:=	Project_Infomation.Major;
ht_CAN4_8DD1_Tx.Data[3]		:=	Project_Infomation.Minor;
ht_CAN4_8DD1_Tx.Data[4]		:=	Project_Infomation.Patch;// Patch
ht_CAN4_8DD1_Tx.Data[5].0	:=	0; // Buzzer
ht_CAN4_8DD1_Tx.Data[5].1	:=	0; //Body Not Ready
ht_CAN4_8DD1_Tx.Data[5].2	:=	0; //Caps Discharging
ht_CAN4_8DD1_Tx.Data[5].3	:=	gq_Allison_Pad_Override	; 
ht_CAN4_8DD1_Tx.Data[5].4	:=	gq_Sevcon_ePTO_Installed;
ht_CAN4_8DD1_Tx.Data[5].5	:=	0;
ht_CAN4_8DD1_Tx.Data[5].6	:=	0;
ht_CAN4_8DD1_Tx.Data[5].7	:=	0;
ht_CAN4_8DD1_Tx.Data[6]	:=	0;
ht_CAN4_8DD1_Tx.Data[7]	:=	0;
ht_CAN4_8DD1_Tx.Len		:=	8;

(***************************************************************************)
ht_CAN4_601_Tx.ID		:=	16#601;
ht_CAN4_601_Tx.Data[0]	:=	UINT_TO_USINT(CAN4_TxConversion.gu16_CAN4_TripCounter_km_Tx);
ht_CAN4_601_Tx.Data[1]	:=	UINT_TO_USINT(SHR(CAN4_TxConversion.gu16_CAN4_TripCounter_km_Tx, 8));
ht_CAN4_601_Tx.Data[2]	:=	SINT_TO_USINT(CAN4_TxConversion.gs8_CAN4_CruiseControlSetpoint_Tx);
ht_CAN4_601_Tx.Data[3]	:=	INT_TO_USINT(CAN4_TxConversion.gs16_CAN4_PowerIndication_Tx);
ht_CAN4_601_Tx.Data[4]	:=	INT_TO_USINT(SHR(CAN4_TxConversion.gs16_CAN4_PowerIndication_Tx, 8));
ht_CAN4_601_Tx.Data[5]	:=	SINT_TO_USINT(CAN4_TxConversion.gs8_CAN4_DummyScreen601_Tx);		
ht_CAN4_601_Tx.Data[6]	:=	0;		
ht_CAN4_601_Tx.Data[7]	:=	0;		
ht_CAN4_601_Tx.Len		:=	8;

ht_CAN4_201_Tx.ID		:=	16#201;
ht_CAN4_201_Tx.Data[0]	:=	SINT_TO_USINT(CAN4_TxConversion.gs8_CAN4_DisplayTemp_Tx);
ht_CAN4_201_Tx.Data[1]	:=	SINT_TO_USINT(CAN4_TxConversion.gs8_CAN4_DisplayDirection_Tx);
ht_CAN4_201_Tx.Data[2]	:=	SINT_TO_USINT(CAN4_TxConversion.gs8_CAN4_SOC_Tx);
ht_CAN4_201_Tx.Data[3]	:=	SINT_TO_USINT(CAN4_TxConversion.gs8_CAN4_DispVehicleStatus_Tx);
ht_CAN4_201_Tx.Data[4]	:=	SINT_TO_USINT(CAN4_TxConversion.gs8_CAN4_PowerIndicationRelative_Tx);
ht_CAN4_201_Tx.Data[5]	:=	SINT_TO_USINT(CAN4_TxConversion.gs8_CAN4_DisplayStatus_Tx);
ht_CAN4_201_Tx.Data[6]	:=	SINT_TO_USINT(CAN4_TxConversion.gs8_CAN4_SOC1_Tx);
ht_CAN4_201_Tx.Data[7]	:=	SINT_TO_USINT(CAN4_TxConversion.gs8_CAN4_BatteryVoltage_Tx);
ht_CAN4_201_Tx.Len		:=	8;

ht_CAN4_301_Tx.ID		:=	16#301;
ht_CAN4_301_Tx.Data[0]	:=	INT_TO_USINT(CAN4_TxConversion.gs16_CAN4_BatteryCurrent_Tx);
ht_CAN4_301_Tx.Data[1]	:=	INT_TO_USINT(SHR(CAN4_TxConversion.gs16_CAN4_BatteryCurrent_Tx, 8));
ht_CAN4_301_Tx.Data[2]	:=	UINT_TO_USINT(CAN4_TxConversion.gu16_CAN4_DisplayRangeMin_Tx);
ht_CAN4_301_Tx.Data[3]	:=	UINT_TO_USINT(SHR(CAN4_TxConversion.gu16_CAN4_DisplayRangeMin_Tx, 8));
ht_CAN4_301_Tx.Data[4]	:=	UINT_TO_USINT(gu16_BMS1_LowCellVoltage); (*gu8_BMS1_LowCellV_Tx*)
ht_CAN4_301_Tx.Data[5]	:=	UINT_TO_USINT(SHR(gu16_BMS1_LowCellVoltage, 8)); (*gu8_BMS2_LowCellV_Tx*)
ht_CAN4_301_Tx.Data[6]	:=	UINT_TO_USINT(gu16_BMS2_LowCellVoltage);
ht_CAN4_301_Tx.Data[7]	:=	UINT_TO_USINT(SHR(gu16_BMS2_LowCellVoltage, 8));
ht_CAN4_301_Tx.Len		:=	8;

ht_CAN4_401_Tx.ID		:=	16#401;
ht_CAN4_401_Tx.Data[0]	:=	SINT_TO_USINT(CAN4_TxConversion.gs8_CAN4_MotorTemp_Tx);
ht_CAN4_401_Tx.Data[1]	:=	SINT_TO_USINT(CAN4_TxConversion.gs8_CAN4_InverterTemp_Tx);
ht_CAN4_401_Tx.Data[2]	:=	CAN4_TxConversion.gu8_CAN4_ChargerStatus_Tx;
ht_CAN4_401_Tx.Data[3]	:=	SINT_TO_USINT(CAN4_TxConversion.gs8_CAN4_ThrottlePedal_Tx);
ht_CAN4_401_Tx.Data[4]	:=	16#ff;
ht_CAN4_401_Tx.Data[5]	:=	SINT_TO_USINT(CAN4_TxConversion.gs8_CAN4_VehicleSpeedMsg_Tx);
ht_CAN4_401_Tx.Data[6]	:=	SINT_TO_USINT(CAN4_TxConversion.gs8_CAN4_VehicleStatus_Tx);
ht_CAN4_401_Tx.Data[7]	:=	SINT_TO_USINT(CAN4_TxConversion.gs8_CAN4_RegenTorquePercDisplay_Tx);
ht_CAN4_401_Tx.Len		:=	8;
(***************************************************************************)


ht_ETC2_Tx.ID		:=	16#18F00503 OR EPEC_CANVXD.MASK_29BIT;
ht_ETC2_Tx.Data[0]	:=	gu8_CurrentGear2; (*Current Gear2*)
ht_ETC2_Tx.Data[1]	:=	UINT_TO_USINT(gu16_CurrentGear); (*Current Gear LSB*)
ht_ETC2_Tx.Data[2]	:=	UINT_TO_USINT(SHR(gu16_CurrentGear, 8)); (*Current Gear MSB*)
ht_ETC2_Tx.Data[3]	:=	gu8_CurrentGear2; (*Current Gear2*)
ht_ETC2_Tx.Data[4]	:=	16#FF;
ht_ETC2_Tx.Data[5]	:=	16#FF;
ht_ETC2_Tx.Data[6]	:=	UINT_TO_USINT(gu16_CurrentGear1); (*Current Gear1 LSB*)
ht_ETC2_Tx.Data[7]	:=	UINT_TO_USINT(SHR(gu16_CurrentGear1, 8)); (*Current Gear1 MSB*)
ht_ETC2_Tx.Len		:=	8;

NMT1_Tx.ID		:=	0;
NMT1_Tx.Data[0]	:=	1;
NMT1_Tx.Data[1]	:=	0;
NMT1_Tx.Len		:=	2;

Dash_FF08_Tx.ID	:=	16#18FF08C4 OR EPEC_CANVXD.MASK_29BIT;
Dash_FF08_Tx.Data[0].0	:=	DO_q_DrivetrainCoolingFan_DO;
Dash_FF08_Tx.Data[0].1	:=	gq_Dash_Sevcon1_Enable;
Dash_FF08_Tx.Data[0].2	:=	gq_Dash_Sevcon2_Enable;
Dash_FF08_Tx.Data[0].3	:=	DO_q_DrivetrainDCDCInhibit_DO;
Dash_FF08_Tx.Data[0].4	:=	Brusa1_Rx.S_ProximityDet;
Dash_FF08_Tx.Data[0].5	:=	DO_q_Battery1ChargePrecharge_DO;
Dash_FF08_Tx.Data[0].6	:=	DO_q_Battery1ChargeMain_DO;
Dash_FF08_Tx.Data[0].7	:=	DO_q_Battery2ChargePrecharge_DO;
Dash_FF08_Tx.Data[1].0	:=	DO_q_Battery2ChargeMain_DO;
Dash_FF08_Tx.Data[1].1	:=	gq_Dash_Charge_Rq;
Dash_FF08_Tx.Data[1].2	:=	gq_Dash_Discharge_Rq;
Dash_FF08_Tx.Data[1].3	:=	gq_Dash_Charge_Rq;
Dash_FF08_Tx.Data[1].4	:=	gq_Dash_Discharge_Rq;
Dash_FF08_Tx.Data[1].5	:=	DI_q_VehicleKL15_DI;
Dash_FF08_Tx.Data[1].6	:=	(Brusa.LEDDem = Brusa.LED_RED);//DO_q_ChargePlugLED_Red_DO;
Dash_FF08_Tx.Data[1].7	:=	(Brusa.LEDDem = Brusa.LED_GREEN);//DO_q_ChargePlugLED_Green_DO;
Dash_FF08_Tx.Data[2]	:=	gu8_SystemState; (*Might need to change this*)
Dash_FF08_Tx.Data[3]	:=	REAL_TO_USINT(gr_VehicleSpeed_kmph);
Dash_FF08_Tx.Data[4]	:=	gu8_BMS_SOC;
Dash_FF08_Tx.Data[5]	:=	INT_TO_USINT(gs16_Dash_BattCurrent_Tx);
Dash_FF08_Tx.Data[6]	:=	INT_TO_USINT(SHR(gs16_Dash_BattCurrent_Tx, 8));
Dash_FF08_Tx.Data[7].0	:=	DO_q_BatteryDischargePrecharge_DO;
Dash_FF08_Tx.Data[7].1	:=	DO_q_BatteryDischargeMain_DO;
Dash_FF08_Tx.Len	:=	8;

Dash_FF12_Tx.ID	:=	16#18FF12C4 OR EPEC_CANVXD.MASK_29BIT;
Dash_FF12_Tx.Data[0].0	:=	DI_q_VehicleKL15_DI;
Dash_FF12_Tx.Data[0].1	:=	FALSE; (*Crawl*)
Dash_FF12_Tx.Data[0].2	:=	gq_BrakeSwitch;
Dash_FF12_Tx.Data[0].3	:=	gq_HandBrake;
Dash_FF12_Tx.Data[0].4	:=	gq_BattFullyCharged;
Dash_FF12_Tx.Data[0].5	:=	HMI_Rx.Heater_Enable;
Dash_FF12_Tx.Data[0].6	:=	FALSE; (*DI AC*)
Dash_FF12_Tx.Data[0].7	:=	((Brusa.LEDDem = Brusa.LED_BLUE) OR (Brusa.LEDDem = (Brusa.LED_BLUE AND Brusa.LED_GREEN_PULSE)));//DO_q_ChargePlugLED_Blue_DO;
Dash_FF12_Tx.Data[1]	:=	gu8_CurrentGear2;
Dash_FF12_Tx.Data[2]	:=	gu8_Dash_AccelPedal_Tx;
Dash_FF12_Tx.Data[3]	:=	hu8_Temp; (*Inverter Temp*)
Dash_FF12_Tx.Data[4]	:=	gu8_Dash_BrakePressure1_Tx;
Dash_FF12_Tx.Data[5]	:=	gu8_Dash_BrakePressure2_Tx;
Dash_FF12_Tx.Data[6]	:=	INT_TO_USINT(gs16_Dash_Power);
Dash_FF12_Tx.Data[7]	:=	INT_TO_USINT(SHR(gs16_Dash_Power, 8));
Dash_FF12_Tx.Len	:=	8;
(*
(*BMS*)
Dash_FF02_Tx.ID	:=	16#18FF02C4;
Dash_FF02_Tx.Data[0]	:=	REAL_TO_USINT(gr_BMS_BatteryVoltage);
Dash_FF02_Tx.Data[1]	:=	UINT_TO_USINT(SHR(REAL_TO_UINT(gr_BMS_BatteryVoltage), 8));
Dash_FF02_Tx.Data[2]	:=	UINT_TO_USINT(gu16_BMS1_LowCellVoltage);
Dash_FF02_Tx.Data[3]	:=	UINT_TO_USINT(SHR(gu16_BMS1_LowCellVoltage, 8));
Dash_FF02_Tx.Data[4]	:=	UINT_TO_USINT(gu16_BMS1_HighCellVoltage);
Dash_FF02_Tx.Data[5]	:=	UINT_TO_USINT(SHR(gu16_BMS1_HighCellVoltage, 8));
Dash_FF02_Tx.Data[6]	:=	UINT_TO_USINT(gu16_BMS1_LowCellVoltage_ID);
Dash_FF02_Tx.Data[7]	:=	UINT_TO_USINT(gu16_BMS1_HighCellVoltage_ID);
Dash_FF02_Tx.Len	:=	8;
Dash_FF04_Tx.ID	:=	16#18FF04C4;
Dash_FF04_Tx.Data[0]	:=	REAL_TO_USINT(gr_BMS_DCL);
Dash_FF04_Tx.Data[1]	:=	UINT_TO_USINT(SHR(REAL_TO_UINT(gr_BMS_DCL), 8));
Dash_FF04_Tx.Data[2]	:=	INT_TO_USINT(gs16_BMS_BatteryCurrent);
Dash_FF04_Tx.Data[3]	:=	INT_TO_USINT(SHR(REAL_TO_INT(gs16_BMS_BatteryCurrent), 8));
Dash_FF04_Tx.Data[4]	:=	REAL_TO_USINT(gr_BMS1_Voltage);
Dash_FF04_Tx.Data[5]	:=	UINT_TO_USINT(SHR(REAL_TO_UINT(gr_BMS1_Voltage), 8));
Dash_FF04_Tx.Data[6]	:=	REAL_TO_USINT(gr_BMS_CCL);
Dash_FF04_Tx.Data[7]	:=	UINT_TO_USINT(SHR(REAL_TO_UINT(gr_BMS_CCL), 8));
Dash_FF04_Tx.Len	:=	8;
Dash_FF21_Tx.ID	:=	16#18FF21C4;
Dash_FF21_Tx.Data[0]	:=	gu8_BMS_LowTemp_ID;
Dash_FF21_Tx.Data[1]	:=	gu8_BMS_HighTemp_ID;
Dash_FF21_Tx.Data[2]	:=	SINT_TO_USINT(gs8_Dash_AverageTemp_Tx);
Dash_FF21_Tx.Data[3]	:=	SINT_TO_USINT(gs8_Dash_HighTemp_Tx);
Dash_FF21_Tx.Data[4]	:=	SINT_TO_USINT(gs8_Dash_LowTemp_Tx);
Dash_FF21_Tx.Data[5]	:=	gu8_BMS_SOC;
Dash_FF21_Tx.Data[6]	:=	0;
Dash_FF21_Tx.Data[7]	:=	0;
Dash_FF21_Tx.Len	:=	8;	
*)

Dash_FF14_Tx.ID	:=	16#18FF14C4 OR EPEC_CANVXD.MASK_29BIT;
Dash_FF14_Tx.Data[0]	:=	INT_TO_USINT(gs16_Sevcon1_SpeedMeasured);
Dash_FF14_Tx.Data[1]	:=	INT_TO_USINT(SHR(gs16_Sevcon1_SpeedMeasured, 8));
Dash_FF14_Tx.Data[2]	:=	INT_TO_USINT(gs16_Sevcon2_SpeedMeasured);
Dash_FF14_Tx.Data[3]	:=	INT_TO_USINT(SHR(gs16_Sevcon2_SpeedMeasured, 8));
Dash_FF14_Tx.Data[5]	:=	REAL_TO_USINT(gr_Sevcon1_DCLink_Voltage);
Dash_FF14_Tx.Data[4]	:=	UINT_TO_USINT(SHR(REAL_TO_UINT(gr_Sevcon1_DCLink_Voltage * 16), 8));
Dash_FF14_Tx.Data[7]	:=	REAL_TO_USINT(gr_Sevcon2_DCLink_Voltage);
Dash_FF14_Tx.Data[6]	:=	UINT_TO_USINT(SHR(REAL_TO_UINT(gr_Sevcon2_DCLink_Voltage  *16), 8));
Dash_FF14_Tx.Len	:=	8;

CAN4_HMI_Tx.ID    := 16#18BB3244 OR EPEC_CANVXD.MASK_29BIT;
CAN4_HMI_Tx.Data[0]  := Brusa.chargeStatus;
CAN4_HMI_Tx.Data[1]  := 0;
CAN4_HMI_Tx.Data[2]  := 0;
CAN4_HMI_Tx.Data[3]  := 0;
CAN4_HMI_Tx.Data[4]  := 0;
CAN4_HMI_Tx.Data[5]  := 0;
CAN4_HMI_Tx.Data[6]  := 0;
CAN4_HMI_Tx.Len   := 8;
(*FA00 new address to start on, choose an appropriate source address for the controller*)


hton_MessageSend_Timer(IN := NOT(hton_MessageSend_Timer.Q), PT := T#100MS);
IF (hton_MessageSend_Timer.Q = TRUE) THEN
	G_CAN4_Channel.SendMessage(i_pMSG:=ADR(ht_ETC2_Tx));
	(*Dash Screen*)
	G_CAN4_Channel.SendMessage(i_pMSG:=ADR(Dash_FF08_Tx));
	G_CAN4_Channel.SendMessage(i_pMSG:=ADR(Dash_FF12_Tx));
	G_CAN4_Channel.SendMessage(i_pMSG:=ADR(Dash_FF14_Tx));
	
	(*G_CAN4_Channel.SendMessage(i_pMSG:=ADR(Dash_FF08_Tx));
	G_CAN4_Channel.SendMessage(i_pMSG:=ADR(Dash_FF04_Tx));
	G_CAN4_Channel.SendMessage(i_pMSG:=ADR(Dash_FF02_Tx));
	G_CAN4_Channel.SendMessage(i_pMSG:=ADR(Dash_FF21_Tx));*)

END_IF
Tx_Timer(IN := NOT(Tx_Timer.Q), PT := T#1000MS);
IF (Tx_Timer.Q = TRUE) THEN
	G_CAN4_Channel.SendMessage(i_pMSG:=ADR(NMT1_Tx));
	
	G_CAN4_Channel.SendMessage(i_pMSG:=ADR(CAN4_HMI_Tx));
	G_CAN4_Channel.SendMessage(i_pMSG:=ADR(ht_CAN4_601_Tx));
	G_CAN4_Channel.SendMessage(i_pMSG:=ADR(ht_CAN4_201_Tx));
	G_CAN4_Channel.SendMessage(i_pMSG:=ADR(ht_CAN4_301_Tx));
	G_CAN4_Channel.SendMessage(i_pMSG:=ADR(ht_CAN4_401_Tx));
	G_CAN4_Channel.SendMessage(i_pMSG:=ADR(ht_CAN4_8DD1_Tx));
	
END_IF

END_PROGRAM

// Application/UserCode/CAN4/CAN4_TxConversion_1
PROGRAM CAN4_TxConversion_1
VAR
	(*Vehicle Direction (FORWARD := 16#7E, NEUTRAL := 16#7D, REVERSE := 16#7C, UNKNOWN := 16#00)*)
	(*********************************************)
	(*601*)
	gu16_CAN4_TripCounter_km_Tx			:	UINT;
	gu16_CAN4_DisplayRangeMin_Tx		:	UINT;
	gu16_CAN4_DisplayRangeMax_Tx		:	UINT;
	gu16_CAN4_DisplayRangeEst_Tx		:	UINT;
	(*201*)
	gs8_CAN4_CruiseControlSetpoint_Tx	:	SINT;
	gs8_CAN4_DummyScreen601_Tx			:	SINT;
	gs8_CAN4_DisplayTemp_Tx				:	SINT;
	gs8_CAN4_DisplayDirection_Tx		:	SINT;
	gs8_CAN4_SOC_Tx						:	SINT;
	gs8_CAN4_DispVehicleStatus_Tx		:	SINT;
	gs8_CAN4_PowerIndicationRelative_Tx	:	SINT;
	gs8_CAN4_DisplayStatus_Tx			:	SINT;
	(*301*)
	gs8_CAN4_SOC1_Tx					:	SINT;
	gs8_CAN4_BatteryVoltage_Tx			:	SINT;
	gs8_CAN4_MotorTemp_Tx				:	SINT;
	gs8_CAN4_InverterTemp_Tx			:	SINT;
	gu8_CAN4_ChargerStatus_Tx			:	USINT;
	gq_CAN4_ChargerPP_Tx				:	BOOL;
	gs8_CAN4_ThrottlePedal_Tx			:	SINT;
	gs8_CAN4_BrakePedal_Tx				:	SINT;
	gs8_CAN4_VehicleSpeedMsg_Tx			:	SINT;
	(*401*)
	gs8_CAN4_VehicleStatus_Tx			:	SINT;
	gs8_CAN4_RegenTorquePercDisplay_Tx	:	SINT;
	gs16_CAN4_PowerIndication_Tx		:	INT;
	gs16_CAN4_BatteryCurrent_Tx			:	INT;
	
	(*********************************************)
	

END_VAR
VAR CONSTANT
	DISPLAY_EST_RANGE_OFFSET	:	USINT	:=	10;
	DISPLAY_EST_RANGE_CF	:	USINT	:=	3;
	BATTERY_VOLTAGE_DISPLAY_CF	:	REAL	:=	0.25;
	DISPLAY_POWER_CF	:	UINT	:=	1000;
	DISPLAY_POWER_OFFSET	:	UINT	:=	32768;
	CHARGER_DETECTED	:	USINT	:=	0;
	
	
END_VAR


IF (gq_Gear_Neutral = TRUE) THEN
	gu16_CurrentGear	:=	0;
	gu16_CurrentGear1	:=	16#204E;
	gu8_CurrentGear2	:=	16#7D;
ELSIF (gq_Gear_Drive = TRUE) THEN
	gu16_CurrentGear	:=	16#2941;
	gu16_CurrentGear1	:=	16#2044;
	gu8_CurrentGear2	:=	16#7E;
ELSIF (gq_Gear_Reverse = TRUE) THEN
	gu16_CurrentGear	:=	16#2941;
	gu16_CurrentGear1	:=	16#2052;
	gu8_CurrentGear2	:=	16#7C;
END_IF

IF (Brusa1_Rx.StatusPP = CHARGER_DETECTED) THEN
	gq_CAN4_ChargerPP_Tx	:=	TRUE;
ELSE
	gq_CAN4_ChargerPP_Tx	:=	FALSE;
END_IF


(*601*)
gu16_CAN4_TripCounter_km_Tx			:=	00; (*0*)
gu16_CAN4_DisplayRangeMin_Tx		:=	00; (*0*)
gu16_CAN4_DisplayRangeMax_Tx		:=	00; (*0*)
gu16_CAN4_DisplayRangeEst_Tx		:=	LIMIT(0, (gu8_BMS_SOC - DISPLAY_EST_RANGE_OFFSET), 100) * DISPLAY_EST_RANGE_CF;
(*201*)
gs8_CAN4_CruiseControlSetpoint_Tx	:=	00; (*Need to add this when cruise control added*)
gs8_CAN4_DummyScreen601_Tx			:=	00; (*Need to find out what this is used for*)
gs8_CAN4_DisplayTemp_Tx				:=	INT_TO_SINT(gs16_MaxTemp_degC);
gs8_CAN4_DisplayDirection_Tx		:=	00; (*Bits*)
gs8_CAN4_DisplayDirection_Tx.3		:=	FALSE; // ePTO active to go here.
gs8_CAN4_DisplayDirection_Tx.4		:=	gq_Gear_Drive;
gs8_CAN4_DisplayDirection_Tx.5		:=	gq_Gear_Reverse;
gs8_CAN4_DisplayDirection_Tx.6		:=	gq_Gear_Neutral;
gs8_CAN4_DisplayDirection_Tx.7		:=	gq_HandBrake;
gs8_CAN4_SOC_Tx						:=	USINT_TO_SINT(gu8_BMS_SOC); (*SOC*)

gs8_CAN4_DisplayStatus_Tx.0		:=	00;
gs8_CAN4_DisplayStatus_Tx.1		:=	00;
gs8_CAN4_DisplayStatus_Tx.2		:=	DI_q_Aux_Pos_Discharge_Master_DI; (*Aux Pos Cont 1*)
gs8_CAN4_DisplayStatus_Tx.3		:=	DI_q_Aux_Neg_Discharge_Master_DI; (*Aux Neg Cont 1*)
gs8_CAN4_DisplayStatus_Tx.4		:=	DI_q_Aux_Pos_Discharge_Slave_DI; (*Aux Pos Cont 2*)
gs8_CAN4_DisplayStatus_Tx.5		:=	DI_q_Aux_Neg_Discharge_Slave_DI; (*Aux Neg Cont 2*)
gs8_CAN4_DisplayStatus_Tx.6		:=	gq_EStop; (*E Stop*)
gs8_CAN4_DisplayStatus_Tx.7		:=	gq_EStopLatch; (*E Stop Latch*)

gs8_CAN4_PowerIndicationRelative_Tx	:=	00; (*0*)
gs8_CAN4_DispVehicleStatus_Tx		:=	00; (*Bits, never set*)
(*301*)
gs8_CAN4_SOC1_Tx					:=	USINT_TO_SINT(gu8_BMS_SOC); (*SOC*)
gs8_CAN4_BatteryVoltage_Tx			:=	REAL_TO_SINT(gr_BMS_BatteryVoltage * BATTERY_VOLTAGE_DISPLAY_CF);
gs8_CAN4_MotorTemp_Tx				:=	REAL_TO_SINT(gr_MCU_ThermalIndicator); (*0*)
gs8_CAN4_InverterTemp_Tx			:=	REAL_TO_SINT(gr_MCU_ThermalIndicator); (*MCU Temp*)
gu8_CAN4_ChargerStatus_Tx.0			:=	00; (*0*)
gu8_CAN4_ChargerStatus_Tx.1			:=	00; (*0*)
gu8_CAN4_ChargerStatus_Tx.2			:=	00; (*0*)
gu8_CAN4_ChargerStatus_Tx.3			:=	gq_CAN4_ChargerPP_Tx; (*0*)
gu8_CAN4_ChargerStatus_Tx.4			:=	00; (*0*)
gu8_CAN4_ChargerStatus_Tx.5			:=	00; (*0*)
gu8_CAN4_ChargerStatus_Tx.6			:=	00; (*0*)
gu8_CAN4_ChargerStatus_Tx.7			:=	00; (*0*)
gs8_CAN4_ThrottlePedal_Tx			:=	REAL_TO_SINT(gr_AccelPedal_Perc * 100); (*Throttle Pedal*)
gs8_CAN4_BrakePedal_Tx				:=	00; (*0*)
gs8_CAN4_VehicleSpeedMsg_Tx			:=	00; (*0*)
(*401*)
gs8_CAN4_VehicleStatus_Tx			:=	00; (*Bits, never set*)
gs8_CAN4_VehicleStatus_Tx.1			:=	00; (*Door Open*)
gs8_CAN4_VehicleStatus_Tx.2			:=	00; (*Dashboard Illuminated*)
gs8_CAN4_VehicleStatus_Tx.3			:=	00; (*Power Steering*)
gs8_CAN4_VehicleStatus_Tx.4			:=	00; (*Air Compressor*)
gs8_CAN4_RegenTorquePercDisplay_Tx	:=	00; (*Scaled regen torque*)
gs16_CAN4_PowerIndication_Tx		:=	REAL_TO_INT((ABS(gr_BMS_BatteryVoltage * gs16_BMS_BatteryCurrent) / DISPLAY_POWER_CF) + DISPLAY_POWER_OFFSET); (*(current * batteryVoltage)*-1/1000)+32768*)
gs16_CAN4_BatteryCurrent_Tx			:=	gs16_BMS_BatteryCurrent; (*Current*)

IF (gu16_Sevcon1_Controlword = 5) THEN
	gq_Dash_Sevcon1_Enable	:=	TRUE;
ELSE
	gq_Dash_Sevcon1_Enable	:=	FALSE;
END_IF
IF (gu16_Sevcon2_Controlword = 5) THEN
	gq_Dash_Sevcon2_Enable	:=	TRUE;
ELSE
	gq_Dash_Sevcon2_Enable	:=	FALSE;
END_IF
IF (gu8_SystemState = DRIVE_SYS) THEN
	gq_Dash_Charge_Rq		:=	FALSE;
	gq_Dash_Discharge_Rq	:=	TRUE;
ELSIF (gu8_SystemState = PLUGIN_SYS) THEN
	gq_Dash_Charge_Rq		:=	TRUE;
	gq_Dash_Discharge_Rq	:=	FALSE;
ELSE
	gq_Dash_Charge_Rq		:=	FALSE;
	gq_Dash_Discharge_Rq	:=	FALSE;
END_IF
gs16_Dash_BattCurrent_Tx	:=	gs16_BMS_BatteryCurrent * 10;

IF (gu8_BMS_SOC >= 100 AND gs16_BMS1_CCL <= 0 AND gs16_BMS2_CCL <= 0) THEN
	gq_BattFullyCharged	:=	TRUE;
ELSE
	gq_BattFullyCharged	:=	FALSE;
END_IF

gu8_Dash_AccelPedal_Tx	:=	REAL_TO_USINT(gr_AccelPedal_Perc * 2.5);
gu8_Dash_BrakePressure1_Tx	:=	REAL_TO_USINT(gr_J1939_ServiceBrakeAirPressCircuit1 * 10);
gu8_Dash_BrakePressure2_Tx	:=	REAL_TO_USINT(gr_J1939_ServiceBrakeAirPressCircuit2 * 10);

gs16_Dash_Power	:=	REAL_TO_INT(gr_BMS_BatteryVoltage * gs16_BMS_BatteryCurrent * 0.001);

END_PROGRAM

// Application/UserCode/Contactor Control/ContactorControl_1
PROGRAM ContactorControl_1
VAR
	hton_Precharge_Timer				:	TON;
	hton_PrechargeDisconnect_Timer		:	TON;
	hton_PrechargeDisconnectBMS1_Timer	:	TON;
	hton_PrechargeDisconnectBMS2_Timer	:	TON;
	hton_MainContactorConnection_Delay	:	TON;
	hton_Contactor_Delay				:	TON;
	hr_MainConnectionVoltage			:	REAL;
	hq_BatteryDischargePrecharge_Rq	:	BOOL;
	hq_BatteryDischargeMain_Rq			:	BOOL	:=	FALSE;
	hq_Battery1ChargePrecharge_Rq		:	BOOL;
	hq_Battery1ChargeMain_Rq			:	BOOL;
	hq_Battery2ChargePrecharge_Rq		:	BOOL;
	hq_Battery2ChargeMain_Rq			:	BOOL;
END_VAR

VAR CONSTANT
	CURRENT_DISCONNECT					:	SINT	:=	10; (*Only disconnect below 10Amps*)
	PRECHARGEEND_VOLTAGE_PERC			:	REAL	:=	0.95;
	CONTACTORSWITCH_CURRENT_LIMIT		:	USINT	:=	3; (*Assigned an intial value of 10A*)
END_VAR


(*Non operational system state*)
(*******************************************************************************************************************)

